SYMBOL_TABLE
"I01"	DB 1	FB 1	// STD - Ilot : DB D'INSTANCE DU FB1
"I02"	DB 2	FB 2	// FACILITY: INSTANCE DB FOR MMC CONTROL (FB2)
"I03"	DB 3	FB 3
"I04"	DB 4	FB 4	// FACILITY: INSTANCE DB FOR COMMUNICATION / DB D'INSTANCE POUR LA COMMUNICATION
"CDIV"	DB 69	DB 69	// FACILITY: DIVERSITIES CODES TABLE / TABLE CODES DIVERSITES
"SFM_DB"	DB 75	FB 20	// Bloque de diagnóstico para Notificar errores de sistema
"SFM_GLOBAL_DB"	DB 76	DB 76	// Bloque de diagnóstico para Notificar errores de sistema
"SFM_PN"	DB 77	DB 77	// PROFINET DIAGNOSTIC FUNCTION EDITING DB FOR IHMP
"SIP1"	DB 89	DB 89	// SIPTOL EXCHANGES DATAS / TABLE D'ECHANGES SIPTOL
"PILE"	DB 90	DB 90	// FACILITY: FIFO STORAGE / PILE DE STOCKAGE
"IDENT"	DB 93	DB 93	// RFID DATAS / IDENTIFIANT DYNAMIQUE
"IBD"	DB 95	DB 95	// FACILITY: DATA BASE DB / DB BASE DE DONNEE
"IIT"	DB 96	DB 96	// FACILITY: PART TABLE / DB TABLE PIECE
"IG"	DB 99	DB 99	// FACILITY: GLOBAL DB / DB GLOBAL
"Z1"	DB 100	FB 100	// ZONE 1: ZONE CONTROL / GESTION ZONE
"Z1A0L"	DB 109	FB 109	// A0 LANCEMENT INSTANCE DATA BLOC / BLOC DE DONNEES INSTANCE A0 LANCEMENT
"Z1A0"	DB 110	FB 110	// A0 MONTAGE INSTANCE DATA BLOC / BLOC DE DONNEES INSTANCE A0 MONTAGE
"Z1A1"	DB 111	FB 111	// A1 OP_BPVAL INSTANCE DATA BLOC / BLOC DE DONNEES INSTANCE A1 OP_BPVAL
"Z1A2"	DB 112	FB 112	// A2 OP_BPVAL INSTANCE DATA BLOC / BLOC DE DONNEES INSTANCE A2 OP_BPVAL
"Z1A0M"	DB 115	FB 115
"Z1B0"	DB 120	FB 120
"Z1B1"	DB 121	FB 121	// B1 OP_BPVAL INSTANCE DATA BLOC / BLOC DE DONNEES INSTANCE B1 OP_BPVAL
"Z1B2"	DB 122	FB 122	// B2 OP_BPVAL INSTANCE DATA BLOC / BLOC DE DONNEES INSTANCE B2 OP_BPVAL
"Z1B3"	DB 123	FB 123	// B3 MONTAGE INSTANCE DATA BLOC / BLOC DE DONNEES INSTANCE B3 MONTAGE
"Z1B4"	DB 124	FB 124	// B4 OP_BIMA INSTANCE DATA BLOC / BLOC DE DONNEES INSTANCE B4 OP_BIMA
"Z1B0M"	DB 125	FB 125
"Z1C0"	DB 130	FB 130	// C0 MONTAGE INSTANCE DATA BLOC / BLOC DE DONNEES INSTANCE C0 MONTAGE
"Z1C1"	DB 131	FB 131	// C1 OP_BPVAL INSTANCE DATA BLOC / BLOC DE DONNEES INSTANCE C1 OP_BPVAL
"Z1D0"	DB 140	FB 140	// D0 MONTAGE INSTANCE DATA BLOC / BLOC DE DONNEES INSTANCE D0 MONTAGE
"Z1D1"	DB 141	FB 141	// D1 OP_BIMA INSTANCE DATA BLOC / BLOC DE DONNEES INSTANCE D1 OP_BIMA
"Z1D2"	DB 142	FB 142	// D2 OP_BIMA INSTANCE DATA BLOC / BLOC DE DONNEES INSTANCE D2 OP_BIMA
"Z1D0R"	DB 143	FB 143	// D0 RECALAGE INSTANCE DATA BLOC / BLOC DE DONNEES INSTANCE D0 RECALAGE
"Z1D0V"	DB 144	FB 144	// DB DE INTANCIA DEL FB 144
"Z1T"	DB 198	DB 198	// ZONE1 : Temps Enveloppe Mouvements
"Z1G"	DB 199	DB 199	// ZONE 1: GLOBAL DB
"Z2"	DB 200	FB 200	// DB DE INSTANCIA FB 200
"Z2LG"	DB 210	FB 210	// DB DE INSTANCIA FB 210
"Z2LG1"	DB 211	FB 211	// DB DE INSTANCIA FB 211
"Z2LD"	DB 220	FB 220	// DB DE INSTANCIA FB 220
"Z2LD1"	DB 221	FB 221	// DB DE INSTANCIA FB 221
"Z2T"	DB 298	DB 298	// ZONE2 : Temps Enveloppe Mouvements
"Z2G"	DB 299	DB 299	// ZONE 2: GLOBAL DB
"DB_DATO_LCB_P0PUP"	DB 601	DB 601	// DB DATOS DEL LECTOR DE CODIGO DE BARRA
"DB_DATO_LCB_B0PUP"	DB 602	DB 602
"DB_DATO_LCB_A0PUPI"	DB 603	DB 603
"ITS0"	DB 1100	FB 1100	// ILOT : DB Instance safety management normal task
"ITSZ1_AU_ES_FZ"	DB 1110	FB 1110	// Z1 : DB D'INSTANCE DU FB 1110
"ITSZ1SOP"	DB 1111	FB 1111	// Z1 : DB D'INSTANCE DU FB 1111
"ITSZ2_AU_ES_FZ"	DB 1120	FB 1120	// Z2 : DB D'INSTANCE DU FB 1120
"ITSZ2SOP"	DB 1121	FB 1121	// Z2 : DB D'INSTANCE DU FB 1121
"TSM"	DB 1279	DB 1279	// ILOT : DB Gestion SAFETY Zone ILOT
"F_GLOBDB"	DB 1300	DB 1300	// F_: F_Global_Data Block
"F00290__D0SB___M11"	DB 1301	FB 1300
"F00284__D0SB___M10"	DB 1302	FB 1300
"F00278__D0SB___M09"	DB 1303	FB 1300
"F00272__D0SB___M08"	DB 1304	FB 1300
"F00013_Z1ZBM06"	DB 1314	FB 1300
"F00019_Z1ZBM07"	DB 1315	FB 1300
"F00304_D0A2"	DB 1316	FB 1300
"F00074_M08"	DB 1318	FB 1300
"F00080_M09"	DB 1319	FB 1300
"F00086_M10"	DB 1320	FB 1300
"F00092_M11"	DB 1321	FB 1300
"F00044_M08"	DB 1322	FB 1300
"F00050_M09"	DB 1323	FB 1300
"F00056_M10"	DB 1324	FB 1300
"F00062_M11"	DB 1325	FB 1300
"F00506_B0A2"	DB 1326	FB 1300
"F00454_B0A2"	DB 1327	FB 1300
"F00404_A0A2"	DB 1328	FB 1300
"F00552__LGSB_M08"	DB 1329	FB 1300
"F00560__LGSB_M09"	DB 1330	FB 1300
"F00566__LGSB_M10"	DB 1331	FB 1300
"F00572__LGSB_M11"	DB 1332	FB 1300
"F00632__LDSB_M08"	DB 1333	FB 1300
"F00640__LDSB_M09"	DB 1334	FB 1300
"F00650__LDSB_M10"	DB 1335	FB 1300
"F00660__LDSB_M11"	DB 1336	FB 1300
"Z1MPDEV"	DB 1600	DB 1600	// PALABRA PIEZA ESPECIFICA MARCHA VACIO
"AFF"	DB 1863	DB 1863	// SIEBERT DISPLAY STRING STORAGE / ALMACENAMIENTO MENSAJE VISULIZADOR SIEBERT
"DB_IHM_Wincc"	DB 1962	FB 1962
"DB_PN"	DB 2036	FB 2036	// INSTANCE IO PROFINET DB
"0_01_ILOT"	FB 1	FB 1
"0_02_MMC"	FB 2	FB 2	// FACILITY: BACKUP MANAGEMENT AND DATA RESTITUTION ON EXTERNAL MMC CARD
"0_03_XOP"	FB 3	FB 3	// STD - ILOT :  FB Gestion des MOP ou LOP
"FB SECU"	FB 4	FB 4
"test_vieAPI"	FB 13	FB 13
"SFM_FB"	FB 20	FB 20	// Bloque de diagnóstico para Notificar errores de sistema
"1_00_ZONE_1"	FB 100	FB 100	// ZONE1 : zone management
"1_A0_LANCEMENT"	FB 109	FB 109	// A0 LANCEMENT FUNCTION BLOC / SECTION PROGRAMME A0 LANCEMENT
"1_A0_STAGE"	FB 110	FB 110	// ZONE1 : stage A0 management
"1_A1_OPERATOR"	FB 111	FB 111	// ZONE1 : operator A1 management
"1_A2_OPERATOR"	FB 112	FB 112	// ZONE1 : operator A2 management
"1_A0_MARIAGE"	FB 115	FB 115	// A0 MARIAGE FUNCTION BLOC / SECTION PROGRAMME A0 MARIAGE
"1_B0_STAGE"	FB 120	FB 120	// ZONE1 : stage B0 management
"1_B1_OPERATOR"	FB 121	FB 121	// ZONE1 : operator B1 management
"1_B2_OPERATOR"	FB 122	FB 122	// ZONE1 : operator B2 management
"1_B3_GRIPPER"	FB 123	FB 123	// Bloque de funcion GRIPPER B0
"1_B4_OP_BIMA"	FB 124	FB 124	// B4 OP_BIMA FUNCTION BLOC / SECTION PROGRAMME B4 OP_BIMA
"1_B0_MARIAGE"	FB 125	FB 125	// B0 MARIAGE FUNCTION BLOC / SECTION PROGRAMME B0 MARIAGE
"1_C0_STAGE"	FB 130	FB 130	// ZONE1 : stage C0 management
"1_C1_OPERATOR"	FB 131	FB 131	// ZONE1 : operator C1 management
"1_D0_STAGE"	FB 140	FB 140	// ZONE1 : stage D0 management
"1_D1_OPERATOR"	FB 141	FB 141	// ZONE1 : operator D1 management
"1_D2_OPERATOR"	FB 142	FB 142	// ZONE1 : operator D2 management
"1_D0_RECALAGE"	FB 143	FB 143	// D0 RECALAGE FUNCTION BLOC / SECTION PROGRAMME D0 RECALAGE
"1_D0_VISU"	FB 144	FB 144	// D0 VISU FUNCTION BLOC / SECTION PROGRAMME D0 VISU
"F_TON"	FB 185	FB 185	// F_: Timer Switch On Delay
"F_TOF"	FB 186	FB 186	// F_: Timer Switch Off Delay
"2_00_ZONE_2"	FB 200	FB 200	// ZONE2 : zone management
"2_LG_MONTAGE"	FB 210	FB 210	// LG MONTAGE FUNCTION BLOC / SECTION PROGRAMME LG MONTAGE
"2_LG1_OP_BIMA"	FB 211	FB 211	// LG1 OP_BIMA FUNCTION BLOC / SECTION PROGRAMME LG1 OP_BIMA
"2_LD_MONTAGE"	FB 220	FB 220	// LD MONTAGE FUNCTION BLOC / SECTION PROGRAMME LD MONTAGE
"2_LD1_OP_BIMA"	FB 221	FB 221	// LD1 OP_BIMA FUNCTION BLOC / SECTION PROGRAMME LD1
"TR0"	FB 1000	FB 1000	// ZONE 1 : FB Gestion SAFETY opérateur ilot
"TRZ1SOP"	FB 1010	FB 1010	// ZONE 1 : FB Gestion SAFETY SOP de la zone 1
"TRZ1SOPR"	FB 1011	FB 1011	// Gestion SAFETY des SCR
"TN0"	FB 1100	FB 1100	// ILOT: FB Gestion SAFETY ilot
"TSZ1_AU_ES_FZ"	FB 1110	FB 1110	// ZONE 1 : FB Gestion SAFETY Arrêt d'Urgence (AU) de la zone 1
"TSZ1_SOP"	FB 1111	FB 1111	// ZONE 1 : FB Gestion SAFETY de la Mise en Service (MS) de la zone 1
"TNZ1FZ"	FB 1112	FB 1112	// ZONE 1 : FB Gestion SAFETY des Fermeture Zone (FZ) de la zone 1
"TNZ1SOP"	FB 1113	FB 1113
"TNZ1VAR"	FB 1114	FB 1114	// ZONE 1 : FB Gestion SAFETY des Relais De Ligne (RLV) de la zone 1
"TSZ2_AU_ES_FZ"	FB 1120	FB 1120	// ZONE 2 : FB Gestion SAFETY Arrêt d'Urgence (AU) de la zone 2
"TSZ2_SOP"	FB 1121	FB 1121	// ZONE 2 : FB Gestion SAFETY de la Mise en Service (MS) de la zone 2
"F_IO_CGP"	FB 1300	FB 1300
"F_CTRL_1"	FB 1301	FB 1301
"F_CTRL_2"	FB 1302	FB 1302
"F_DIAG_N"	FB 1303	FB 1303	// F_: Diagnosticbuffer Message with non CPU-Stop
"FITON"	FB 1304	FB 1304
"FIACK_GL"	FB 1305	FB 1305
"BFI_DEVERM"	FB 1600	FB 1600	// Gestion du déverminage d'une table
"BF_MID_Ordre"	FB 1602	FB 1602
"DP_locator"	FB 1649	FB 1649
"TUSEND"	FB 1681	FB 1681	// Send Data via UDP
"TCON"	FB 1685	FB 1685	// Connect
"PUT"	FB 1689	FB 1689	// Write Data to a Remote CPU
"GET"	FB 1690	FB 1690	// Read Data From a Remote CPU
"F_SENDDP"	FB 1692	FB 1692	// F_: Send Data via PROFIBUS DP / PROFINET IO
"F_ACK_GL"	FB 1695	FB 1695	// ACKNOWLEDGE OF ALL PERIPHERALS F / ACQUITTEMENT GLOBAL PERIPH F
"P_SEND"	FB 1698	FB 1698	// Send Data to CP340
"P_RCV"	FB 1699	FB 1699	// Receive Data from CP340
"BFS_BSEC1"	FB 1710	FB 1710
"BFS_AIR1"	FB 1713	FB 1713
"BFS_CRM1"	FB 1714	FB 1714
"BFS_BIMA"	FB 1719	FB 1719
"BF_DEVERM"	FB 1803	FB 1803	// BF STAGE DRY RUN CONTROL / BF GESTION DEVERMINAGE POSTE
"BF_CARACT_SIEBERT"	FB 1856	FB 1856	// SIEBERT DISPLAY MESSAGE CONFIGURATION / MISE EN FORME MESSAGE AFFICHEUR SIEBERT
"BF_RECALAGE2"	FB 1857	FB 1857
"BF_LANCEMENT"	FB 1858	FB 1858	// GESTION LANCEMENT SIPTOL
"BF_AFF SIEBERT (2*13) PN"	FB 1860	FB 1860
"BF_CONF_MACHINE"	FB 1869	FB 1869	// GESTION BASE DE DONNEE CONFIGURATION MACHINE
"BF_CODE_PROCESS"	FB 1870	FB 1870	// GESTION BASE DE DONNEE CODE PROCESS
"BF_DATABASE3"	FB 1871	FB 1871	// DATABASE MANAGEMENT / GESTION BASE DE DONNEES
"BF_IHMCR1"	FB 1876	FB 1876	// BF gérant l'IHM du relais non piloté par l'API mais controlé
"BF_IHMCRM1"	FB 1877	FB 1877	// BF gérant l'IHM du relais de controçle raccordement de masse CRM
"BF_CABRS"	FB 1897	FB 1897	// Barcode Reader / Lecteur de code a barre
"BF_IHMAIR1"	FB 1931	FB 1931	// BF - ZONE : Diagnostic du bloc BFS_IHMAIR
"BF_ZONE_MODE_IHM1"	FB 1932	FB 1932	// Safety_V2: Zone HMI Operating _modes management/Gestion IHM et mode de la zone
"BF_IHMCRM"	FB 1942	FB 1942	// BF gérant l'IHM du relais de controçle raccordement de masse CRM
"BF_IHMBSEC"	FB 1944	FB 1944	// BF - Zx : Diagnostic SAFETY BFS_BSEC
"BF_MODBUS TCPIP SLAVE"	FB 1961	FB 1961	// Esclave Modbus sur CP Ethernet
"BF_IHM_WINCC"	FB 1962	FB 1962	// BF- Gestion images WinCC Flexible
"BF_PFLEX_PUP"	FB 1999	FB 1999	// Pupitre de recodage
"BF_MMC"	FB 2000	FB 2000	// Sauvegarde et restitution mémoire sur carte mémoire externe (MMC)
"BF_MARIAGE_API"	FB 2003	FB 2003	// Gestion des Mariages Pièces
"BF_ILOT"	FB 2004	FB 2004	// BF- Gestion info lié à l'installation ( Ilot )
"BF_IDENT"	FB 2015	FB 2015
"BF_ROBOT"	FB 2016	FB 2016	// Interface API <=> Robot Version 1.2a
"BF_TCY_SUIV"	FB 2019	FB 2019
"BF_CPT_PIECE"	FB 2021	FB 2021	// BF- Compteur de pièce
"BF_DIAG_PROFINET"	FB 2036	FB 2036	// BF- Diagnostic PROFINET IO
"BF_TF_TP"	FB 2037	FB 2037	// TRANSFERENCIA DE TABLA DE MEMORIAS PIEZAS
"BF_FIFO"	FB 2039	FB 2039
"BF_MOUV2P1"	FB 2042	FB 2042	// BF- Gestion d'un mouvement à 2 positions
"Ilot"	FB 10000	FB 10000	// STD - ILOT : FB Gestion de l'ilot
"Mmc"	FB 10001	FB 10001	// STD - ILOT : FB Gestion de la sauvegarde des données sur carte MMC
"0_00_XOP"	FB 10002	FB 10002	// STD - ILOT :  FB Gestion des MOP ou LOP
"Zone_1"	FB 10100	FB 10100	// STD - Z1 : FB Gestion de la zone
"Z1_ch_elec_flex"	FB 10101	FB 10101	// STD - Z1 : Traitement du changement d'électrodes groupé pour un périmètre flex
"R1_robot_manut"	FB 10511	FB 10511	// R1_robot_manut
"P0_plateau_2pos"	FB 10530	FB 10530	// P0_Mtg: Plateau 2 positions
"V0_elevat"	FB 10600	FB 10600	// V0_elevat
"0_00_CYCLE_ILOT"	FC 1	FC 1	// FACILITY: CALL OF FACILITY FB
"GRP EXE"	FC 2	FC 2
"0_11_SECU_FERMEE"	FC 11	FC 11	// STD - Recopie des informations SAFETY zones 1 à 9 pour la sécurité zone fermée
"SFM_FC"	FC 22	FC 22	// Bloque de diagnóstico para Notificar errores de sistema
"1_00_cycle Z1"	FC 100	FC 100	// Définition cyclique zone 1
"2_00_cycleZ2"	FC 200	FC 200	// Définition cyclique zone 1
"0_00_TSSAFETY"	FC 1100	FC 1100	// STD - ILOT : Groupe d'exécution F associé à l'OB32 (tâche normale)
"0_00_TSCYCLE"	FC 1101	FC 1101	// ILOT : Appel des FB hors opérateurs liées à l'ILOT
"AG_SEND"	FC 1698	FC 1698	// AG SEND
"AG_RECV"	FC 1699	FC 1699	// AG RECEIVE
"Badi"	I 0.0	BOOL	// [MOP1]   BP ANNULATION DEFAUTS ILOT
"Bri"	I 0.1	BOOL	// [MOP1]  BP REARMEMENT ILOT
"bmcy"	I 0.2	BOOL	// [MOP1] ZONE 1: BP MARCHE CYCLE
"smm"	I 0.3	BOOL	// [MOP1] ZONE 1: SEL. MARCHE MANUELLE REGLAGE
"sma"	I 0.4	BOOL	// [MOP1] ZONE 1: SEL. MARCHE AUTOMATIQUE
"bmr"	I 0.5	BOOL	// [MOP1] ZONE 1: BP MOUVEMENT RETOUR
"bma"	I 0.6	BOOL	// [MOP1] ZONE 1: BP MOUVEMENT ALLER
"Dclim"	I 1.0	BOOL	// [MOP1] DEFAUT CLIM. (Option)
"CCFRO1"	I 10.0	BOOL	// Z1B[M02] Safety Common Control 1(F-RO)
"CCFRO2"	I 10.1	BOOL	// Z1B[M02] Safety Common Control 2(F-RO)
"LG_CB380V"	I 10.2	BOOL	// Z1B[M02] LG CB CONTROL DISJUNTOR 380V MOTOR
"LD_CB380V"	I 10.4	BOOL	// Z1B[M02] LD CB CONTROL DISJUNTOR 380V MOTOR
"CCB24Z"	I 10.6	BOOL	// Z1B[M02] Elec.Circuit Breake 24V(1-24Z)
"CCB24R"	I 10.7	BOOL	// Z1B[M02] Elec.Circuit Breake 24V(1-24R)
"CP7b"	I 11.3	BOOL	// Presostato A0
"Z1CRM"	I 11.4	BOOL	// Z1B[M03] CONTROL RELAY CRM
"SOP_bmcy"	I 11.5	BOOL	// [SOP1] ZONE 1: BP MARCHE CYCLE
"SOP_bmr"	I 11.6	BOOL	// [SOP1] ZONE 1: BP MOUVEMENT RETOUR
"SOP_bma"	I 11.7	BOOL	// [SOP1] ZONE 1: BP MOUVEMENT ALLER
"BAUI"	I 13.0	BOOL	// Z1B[M06] EGS Facility(MOP)
"Z1BAU1"	I 13.1	BOOL	// [SOP1] SOP1 ARRET D'URGENCE ILOT
"SSZ11"	I 13.2	BOOL	// Z1B[M06] SAFETY ZONE SELECTOR ON 1
"BAUL12"	I 13.4	BOOL	// Z1B[M06] EGS Facility(LOP) 2
"SSZ12"	I 13.6	BOOL	// Z1B[M06] SAFETY ZONE SELECTOR ON 2
"Z1_AU_FRO"	I 24.0	BOOL	// Z1B[M08] SAFETY RELAY F-RO AU
"Z1_KMS"	I 25.0	BOOL	// Z1B[M09] SAFETY RELAY F-RO ES
"A0_CCSOP"	I 40.0	BOOL	// A0SB[M02] CONTROL POWER NORMAL SOP
"A0_CCSOPTR"	I 40.1	BOOL	// A0SB[M02] CONTROL POWER NORMAL SOPTR
"A0_CCB24Z"	I 40.4	BOOL	// A0SB[M02] Elec.Circuit Breake 24V(24Z)
"A0_CCB24R"	I 40.5	BOOL	// A0SB[M02] Elec.Circuit Breake 24V(24R)
"A1VAL"	I 41.0	BOOL	// A0SB[M03] A1 OPERATION BOX 1 PB ON VALIDATION
"A2VAL"	I 41.1	BOOL	// A0SB[M03] A2 OPERATION BOX 2 PB ON VALIDATION
"A1CPOP1"	I 50.0	BOOL	// A0SB[M09] Laser scanner 1 NORMAL 1-1 A1
"A2CPOP1"	I 50.1	BOOL	// A0SB[M09] Laser scanner 1 NORMAL 2-1 A2
"A1CPOP2"	I 50.4	BOOL	// A0SB[M09] Laser scanner 1 NORMAL 1-2 A1
"A2CPOP2"	I 50.5	BOOL	// A0SB[M09] Laser scanner 1 NORMAL 2-2 A2
"A1BAU1"	I 56.0	BOOL	// A0SB[M10] OPERATION BOX EGS NORMAL 1 A1
"A2BAU1"	I 56.1	BOOL	// A0SB[M10] OPERATION BOX EGS NORMAL 1 A2
"A1BAU2"	I 56.4	BOOL	// A0SB[M10] OPERATION BOX EGS NORMAL 2 A1
"A2BAU2"	I 56.5	BOOL	// A0SB[M10] OPERATION BOX EGS NORMAL 2 A2
"A0_SOP_FRO"	I 67.0	BOOL	// A0SB[M12] OPERATOR SAFETY STAGE A0
"B0_CCSOP"	I 70.0	BOOL	// B0SB[M02] CONTROL POWER NORMAL SOP
"B0_CCSOPTR"	I 70.1	BOOL	// B0SB[M02] CONTROL POWER NORMAL SOPTR
"B0_CCB24Z"	I 70.4	BOOL	// B0SB[M02] Elec.Circuit Breake 24V(24Z)
"B0_CCB24R"	I 70.5	BOOL	// B0SB[M02] Elec.Circuit Breake 24V(24R)
"B1VAL"	I 71.0	BOOL	// B0SB[M03] B1 OPERATION BOX 1 PB ON VALIDATION
"B2VAL"	I 71.1	BOOL	// B0SB[M03] B2 OPERATION BOX 2 PB ON VALIDATION
"A0DCZA"	I 71.4	BOOL	// B0SB[M03] Detector Guinche A0 Zona A
"A0DCZB"	I 71.5	BOOL	// B0SB[M03] Detector Guinche A0 Zona B
"B0DCZC"	I 71.6	BOOL	// B0SB[M03] Detector Guinche B0 Zona C
"B0DCZB"	I 71.7	BOOL	// B0SB[M03] Detector Guinche B0 Zona B
"B1CPOP1"	I 80.0	BOOL	// B0SB[M09] Laser scanner 1 NORMAL 1-1 B1
"B2CPOP1"	I 80.1	BOOL	// B0SB[M09] Laser scanner 1 NORMAL 2-1 B2
"B3_OP4BP11"	I 80.2	BOOL	// B0SB[M09] GRIPPER T-STAND 1 BUTTON 1 (OP3)
"B3_OP4BP21"	I 80.3	BOOL	// B0SB[M09] GRIPPER T-STAND 1 BUTTON 2 (OP3)
"B1CPOP2"	I 80.4	BOOL	// B0SB[M09] Laser scanner 1 NORMAL 1-2 B1
"B2CPOP2"	I 80.5	BOOL	// B0SB[M09] Laser scanner 1 NORMAL 2-2 B2
"B3_OP4BP12"	I 80.6	BOOL	// B0SB[M09] GRIPPER T-STAND 1 BUTTON 1 (OP3)
"B3_OP4BP22"	I 80.7	BOOL	// B0SB[M09] GRIPPER T-STAND 1 BUTTON 2 (OP3)
"B1BAU1"	I 86.0	BOOL	// B0SB[M10] OPERATION BOX EGS NORMAL 1 B1
"B2BAU1"	I 86.1	BOOL	// B0SB[M10] OPERATION BOX EGS NORMAL 1 B2
"B3BAU11"	I 86.2	BOOL	// B0SB[M10] GRIPPER OPERATION BOX EGS NORMAL 3 B1
"B1BAU2"	I 86.4	BOOL	// B0SB[M10] OPERATION BOX EGS NORMAL 2 B1
"B2BAU2"	I 86.5	BOOL	// B0SB[M10] OPERATION BOX EGS NORMAL 2 B2
"B3BAU12"	I 86.6	BOOL	// B0SB[M10] GRIPPER OPERATION BOX EGS NORMAL 3 B2
"B0_SOP_FRO"	I 97.0	BOOL	// B0SB[M12] OPERATOR SAFETY STAGE B0
"B0_SOP_FRO 2"	I 98.0	BOOL	// B0SB[M13] OPERATOR SAFETY GRIPPER B3
"A0LLS103"	I 100.0	BOOL	// ZONE1 [A0I10] A0 LOCATOR LH X SLIDE ADVANCED
"A0LLS115"	I 100.1	BOOL	// ZONE1 [A0I10] A0 LOCATOR LH X AXIS DETECT 1
"A0LLS117"	I 100.2	BOOL	// ZONE1 [A0I10] A0 LOCATOR LH X AXIS DETECT 3
"A0LLS107"	I 100.3	BOOL	// ZONE1 [A0I10] A0 LOCATOR LH Y SLIDE ADVANCED
"A0LLS104"	I 100.4	BOOL	// ZONE1 [A0I10] A0 LOCATOR LH X SLIDE RETURNED
"A0LLS116"	I 100.5	BOOL	// ZONE1 [A0I10] A0 LOCATOR LH X AXIS DETECT 2
"A0LLS108"	I 100.7	BOOL	// ZONE1 [A0I10] A0 LOCATOR LH Y SLIDE RETURNED
"A0LLS119"	I 101.0	BOOL	// ZONE1 [A0I11] A0 LOCATOR LH Y AXIS DETECT 1
"A0LLS121"	I 101.1	BOOL	// ZONE1 [A0I11] A0 LOCATOR LH Y AXIS DETECT 3
"A0LLS111"	I 101.2	BOOL	// ZONE1 [A0I11] A0 LOCATOR LH Z SLIDE ADVANCED
"A0LLS123"	I 101.3	BOOL	// ZONE1 [A0I11] A0 LOCATOR LH Z AXIS DETECT 1
"A0LLS120"	I 101.4	BOOL	// ZONE1 [A0I11] A0 LOCATOR LH Y AXIS DETECT 2
"A0LLS112"	I 101.6	BOOL	// ZONE1 [A0I11] A0 LOCATOR LH Z SLIDE RETURNED
"A0LLS124"	I 101.7	BOOL	// ZONE1 [A0I11] A0 LOCATOR LH Z AXIS DETECT 2
"A0LLS125"	I 102.0	BOOL	// ZONE1 [A0I12] A0 LOCATOR LH Z AXIS DETECT 3
"A0LS001"	I 102.1	BOOL	// ZONE1 [A0I12] A0 CLAMP ADVANCED
"A0LS004"	I 102.2	BOOL	// ZONE1 [A0I12] A0 CLAMP RETURNED 3
"A0LS002"	I 102.5	BOOL	// ZONE1 [A0I12] A0 CLAMP RETURNED 1
"A0LS008"	I 103.0	BOOL	// ZONE1 [A0I13] A0 L38 GAUGE SWING ADVANCED
"A0LS011"	I 103.2	BOOL	// ZONE1 [A0I13] A0 EJECTOR ADVANCED
"A0LS014"	I 103.3	BOOL	// ZONE1 [A0I13] A0 EJECTOR RETURNED 3
"A0LS009"	I 103.4	BOOL	// ZONE1 [A0I13] A0 L38 GAUGE SWING RETURNED 1
"A0LS012"	I 103.6	BOOL	// ZONE1 [A0I13] A0 EJECTOR RETURNED 1
"A0LS016"	I 104.0	BOOL	// ZONE1 [A0I14] A0 GRIPPER SHIFT 1 ADVANCED
"A0LS018"	I 104.1	BOOL	// ZONE1 [A0I14] A0 GRIPPER SHIFT 2 ADVANCED
"A0LS020"	I 104.2	BOOL	// ZONE1 [A0I14] A0 GRIPPER LOCK 1 ADVANCED
"A0LS017"	I 104.4	BOOL	// ZONE1 [A0I14] A0 GRIPPER SHIFT 1 RETURNED
"A0LS019"	I 104.5	BOOL	// ZONE1 [A0I14] A0 GRIPPER SHIFT 2 RETURNED
"A0LS021"	I 104.6	BOOL	// ZONE1 [A0I14] A0 GRIPPER LOCK 1 RETURNED 1
"A0LS022"	I 104.7	BOOL	// ZONE1 [A0I14] A0 GRIPPER LOCK 1 RETURNED 2
"A0LS024"	I 105.0	BOOL	// ZONE1 [A0I15] A0 GRIPPER LOCK 2 ADVANCED
"A0LS027"	I 105.1	BOOL	// ZONE1 [A0I15] A0 MODEL CHANGE 1 ADVANCED
"A0LS030"	I 105.2	BOOL	// ZONE1 [A0I15] A0 MODEL CHANGE 2 ADVANCED
"A0LS025"	I 105.4	BOOL	// ZONE1 [A0I15] A0 GRIPPER LOCK 2 RETURNED 1
"A0LS028"	I 105.5	BOOL	// ZONE1 [A0I15] A0 MODEL CHANGE 1 RETURNED 1
"A0LS031"	I 105.6	BOOL	// ZONE1 [A0I15] A0 MODEL CHANGE 2 RETURNED 1
"A0LS050"	I 106.0	BOOL	// ZONE1 [A0I16] A0 L38 GRIPPER LH DETECT
"A0LS080"	I 106.2	BOOL	// ZONE1 [A0I16] A0 WORK DETECT 1
"A0LS082"	I 106.3	BOOL	// ZONE1 [A0I16] A0 WORK DETECT 3
"A0LS081"	I 106.6	BOOL	// ZONE1 [A0I16] A0 WORK DETECT 2
"A0LS083"	I 106.7	BOOL	// ZONE1 [A0I16] A0 WORK DETECT 4
"A0RLS103"	I 150.0	BOOL	// ZONE1 [A0I20] A0 LOCATOR RH X SLIDE ADVANCED
"A0RLS115"	I 150.1	BOOL	// ZONE1 [A0I20] A0 LOCATOR RH X AXIS DETECT 1
"A0RLS117"	I 150.2	BOOL	// ZONE1 [A0I20] A0 LOCATOR RH X AXIS DETECT 3
"A0RLS107"	I 150.3	BOOL	// ZONE1 [A0I20] A0 LOCATOR RH Y SLIDE ADVANCED
"A0RLS104"	I 150.4	BOOL	// ZONE1 [A0I20] A0 LOCATOR RH X SLIDE RETURNED
"A0RLS116"	I 150.5	BOOL	// ZONE1 [A0I20] A0 LOCATOR RH X AXIS DETECT 2
"A0RLS108"	I 150.7	BOOL	// ZONE1 [A0I20] A0 LOCATOR RH Y SLIDE RETURNED
"A0RLS119"	I 151.0	BOOL	// ZONE1 [A0I21] A0 LOCATOR RH Y AXIS DETECT 1
"A0RLS121"	I 151.1	BOOL	// ZONE1 [A0I21] A0 LOCATOR RH Y AXIS DETECT 3
"A0RLS111"	I 151.2	BOOL	// ZONE1 [A0I21] A0 LOCATOR RH Z SLIDE ADVANCED
"A0RLS123"	I 151.3	BOOL	// ZONE1 [A0I21] A0 LOCATOR RH Z AXIS DETECT 1
"A0RLS120"	I 151.4	BOOL	// ZONE1 [A0I21] A0 LOCATOR RH Y AXIS DETECT 2
"A0RLS112"	I 151.6	BOOL	// ZONE1 [A0I21] A0 LOCATOR RH Z SLIDE RETURNED
"A0RLS124"	I 151.7	BOOL	// ZONE1 [A0I21] A0 LOCATOR RH Z AXIS DETECT 2
"A0RLS125"	I 152.0	BOOL	// ZONE1 [A0I22] A0 LOCATOR RH Z AXIS DETECT 3
"A0LS005"	I 152.2	BOOL	// ZONE1 [A0I22] A0 CLAMP RETURNED 4
"A0LS007"	I 152.3	BOOL	// ZONE1 [A0I22] A0 CLAMP RETURNED 6
"A0LS003"	I 152.5	BOOL	// ZONE1 [A0I22] A0 CLAMP RETURNED 2
"A0LS006"	I 152.6	BOOL	// ZONE1 [A0I22] A0 CLAMP RETURNED 5
"A0LS015"	I 153.3	BOOL	// ZONE1 [A0I23] A0 EJECTOR RETURNED 4
"A0LS010"	I 153.4	BOOL	// ZONE1 [A0I23] A0 L38 GAUGE SWING RETURNED 2
"A0LS013"	I 153.6	BOOL	// ZONE1 [A0I23] A0 EJECTOR RETURNED 2
"A0LS023"	I 154.4	BOOL	// ZONE1 [A0I24] A0 GRIPPER LOCK 1 RETURNED 3
"A0LS026"	I 154.5	BOOL	// ZONE1 [A0I24] A0 GRIPPER LOCK 2 RETURNED 2
"A0LS029"	I 154.6	BOOL	// ZONE1 [A0I24] A0 MODEL CHANGE 1 RETURNED 2
"A0LS032"	I 154.7	BOOL	// ZONE1 [A0I24] A0 MODEL CHANGE 2 RETURNED 2
"A0LS051"	I 155.0	BOOL	// ZONE1 [A0I25] A0 L38 GRIPPER RH DETECT
"A0LS060"	I 156.0	BOOL	// ZONE1 [A0I26] A0 MANUAL CLAMP RETURNED 1
"A0LS084"	I 156.1	BOOL	// ZONE1 [A0I26] A0 PRESENCIA DE PIEZA EN GABARITO TRASERO
"A0LS061"	I 156.4	BOOL	// ZONE1 [A0I26] A0 MANUAL CLAMP RETURNED 2
"A0LS070"	I 156.7	BOOL	// ZONE1 [A0I26] A0 REMORT SYSTEM IN ZONE DETECT
"B0LLS103"	I 200.0	BOOL	// ZONE1 [B0I10] B0 LOCATOR LH X SLIDE ADVANCED
"B0LLS115"	I 200.1	BOOL	// ZONE1 [B0I10] B0 LOCATOR LH X AXIS DETECT 1
"B0LLS117"	I 200.2	BOOL	// ZONE1 [B0I10] B0 LOCATOR LH X AXIS DETECT 3
"B0LLS107"	I 200.3	BOOL	// ZONE1 [B0I10] B0 LOCATOR LH Y SLIDE ADVANCED
"B0LLS104"	I 200.4	BOOL	// ZONE1 [B0I10] B0 LOCATOR LH X SLIDE RETURNED
"B0LLS116"	I 200.5	BOOL	// ZONE1 [B0I10] B0 LOCATOR LH X AXIS DETECT 2
"B0LLS108"	I 200.7	BOOL	// ZONE1 [B0I10] B0 LOCATOR LH Y SLIDE RETURNED
"B0LLS119"	I 201.0	BOOL	// ZONE1 [B0I11] B0 LOCATOR LH Y AXIS DETECT 1
"B0LLS121"	I 201.1	BOOL	// ZONE1 [B0I11] B0 LOCATOR LH Y AXIS DETECT 3
"B0LLS111"	I 201.2	BOOL	// ZONE1 [B0I11] B0 LOCATOR LH Z SLIDE ADVANCED
"B0LLS123"	I 201.3	BOOL	// ZONE1 [B0I11] B0 LOCATOR LH Z AXIS DETECT 1
"B0LLS120"	I 201.4	BOOL	// ZONE1 [B0I11] B0 LOCATOR LH Y AXIS DETECT 2
"B0LLS112"	I 201.6	BOOL	// ZONE1 [B0I11] B0 LOCATOR LH Z SLIDE RETURNED
"B0LLS124"	I 201.7	BOOL	// ZONE1 [B0I11] B0 LOCATOR LH Z AXIS DETECT 2
"B0LLS125"	I 202.0	BOOL	// ZONE1 [B0I12] B0 LOCATOR LH Z AXIS DETECT 3
"B0LS001"	I 202.1	BOOL	// ZONE1 [B0I12] B0 CLAMP ADVANCED
"B0LS004"	I 202.2	BOOL	// ZONE1 [B0I12] B0 CLAMP RETURNED 3
"B0LS002"	I 202.5	BOOL	// ZONE1 [B0I12] B0 CLAMP RETURNED 1
"B0LS006"	I 202.6	BOOL	// ZONE1 [B0I12] B0 CLAMP RETURNED 5
"B0LS008"	I 203.0	BOOL	// ZONE1 [B0I13] B0 L38 GAUGE SWING ADVANCED
"B0LS011"	I 203.1	BOOL	// ZONE1 [B0I13] B0 EJECTOR ADVANCED
"B0LS014"	I 203.2	BOOL	// ZONE1 [B0I13] B0 EJECTOR RETURNED 3
"B0LS016"	I 203.3	BOOL	// ZONE1 [B0I13] B0 OG SHIFT ADVANCED
"B0LS009"	I 203.4	BOOL	// ZONE1 [B0I13] B0 L38 GAUGE SWING RETURNED 1
"B0LS012"	I 203.5	BOOL	// ZONE1 [B0I13] B0 EJECTOR RETURNED 1
"B0LS017"	I 203.7	BOOL	// ZONE1 [B0I13] B0 OG SHIFT RETURNED
"B0LS018"	I 204.0	BOOL	// ZONE1 [B0I14] B0 OG LOCK ADVANCED
"B0LS020"	I 204.1	BOOL	// ZONE1 [B0I14] B0 OG LOCK RETURNED 2
"B0LS050"	I 204.3	BOOL	// ZONE1 [B0I14] B0 L38 GRIPPER DETECT
"B0LS019"	I 204.4	BOOL	// ZONE1 [B0I14] B0 OG LOCK RETURNED 1
"B0LS021"	I 204.5	BOOL	// ZONE1 [B0I14] B0 OG LOCK RETURNED 3
"B0LS022"	I 205.0	BOOL	// ZONE1 [B0I15] B0 GRIPPER LOCK ADVANCED
"B0LS025"	I 205.1	BOOL	// ZONE1 [B0I15] B0 MODEL CHANGE 1 ADVANCED
"B0LS028"	I 205.2	BOOL	// ZONE1 [B0I15] B0 MODEL CHANGE 2 ADVANCED
"B0LS031"	I 205.3	BOOL	// ZONE1 [B0I15] B0 MODEL CHANGE 3 ADVANCED
"B0LS023"	I 205.4	BOOL	// ZONE1 [B0I15] B0 GRIPPER LOCK RETURNED
"B0LS026"	I 205.5	BOOL	// ZONE1 [B0I15] B0 MODEL CHANGE 1 RETURNED
"B0LS029"	I 205.6	BOOL	// ZONE1 [B0I15] B0 MODEL CHANGE 2 RETURNED 1
"B0LS032"	I 205.7	BOOL	// ZONE1 [B0I15] B0 MODEL CHANGE 3 RETURNED 1
"B0LS080"	I 206.0	BOOL	// ZONE1 [B0I16] B0 WORK DETECT 1
"CP7b_B0"	I 206.3	BOOL	// Presostato - B0
"B0LS081"	I 206.4	BOOL	// ZONE1 [B0I16] B0 WORK DETECT 2
"B0RLS103"	I 250.0	BOOL	// ZONE1 [B0I20] B0 LOCATOR RH X SLIDE ADVANCED
"B0RLS115"	I 250.1	BOOL	// ZONE1 [B0I20] B0 LOCATOR RH X AXIS DETECT 1
"B0RLS117"	I 250.2	BOOL	// ZONE1 [B0I20] B0 LOCATOR RH X AXIS DETECT 3
"B0RLS107"	I 250.3	BOOL	// ZONE1 [B0I20] B0 LOCATOR RH Y SLIDE ADVANCED
"B0RLS104"	I 250.4	BOOL	// ZONE1 [B0I20] B0 LOCATOR RH X SLIDE RETURN
"B0RLS116"	I 250.5	BOOL	// ZONE1 [B0I20] B0 LOCATOR RH X AXIS DETECT 2
"B0RLS108"	I 250.7	BOOL	// ZONE1 [B0I20] B0 LOCATOR RH Y SLIDE RETURNED
"B0RLS119"	I 251.0	BOOL	// ZONE1 [B0I21] B0 LOCATOR RH Y AXIS DETECT 1
"B0RLS121"	I 251.1	BOOL	// ZONE1 [B0I21] B0 LOCATOR RH Y AXIS DETECT 3
"B0RLS111"	I 251.2	BOOL	// ZONE1 [B0I21] B0 LOCATOR RH Z SLIDE ADVANCED
"B0RLS123"	I 251.3	BOOL	// ZONE1 [B0I21] B0 LOCATOR RH Z AXIS DETECT 1
"B0RLS120"	I 251.4	BOOL	// ZONE1 [B0I21] B0 LOCATOR RH Y AXIS DETECT 2
"B0RLS112"	I 251.6	BOOL	// ZONE1 [B0I21] B0 LOCATOR RH Z SLIDE RETURNED
"B0RLS124"	I 251.7	BOOL	// ZONE1 [B0I21] B0 LOCATOR RH Z AXIS DETECT 2
"B0RLS125"	I 252.0	BOOL	// ZONE1 [B0I21] B0 LOCATOR RH Z AXIS DETECT 3
"B0LS005"	I 252.2	BOOL	// ZONE1 [B0I22] B0 CLAMP RETURNED 4
"B0LS003"	I 252.5	BOOL	// ZONE1 [B0I22] B0 CLAMP RETURNED 2
"B0LS007"	I 252.6	BOOL	// ZONE1 [B0I22] B0 CLAMP RETURNED 6
"B0LS010"	I 253.4	BOOL	// ZONE1 [B0I23] B0 L38 GAUGE SWING RETURNED 2
"B0LS013"	I 253.5	BOOL	// ZONE1 [B0I23] B0 EJECTOR RETURNED 2
"B0LS015"	I 253.6	BOOL	// ZONE1 [B0I23] B0 EJECTOR RETURNED 4
"B0LS051"	I 253.7	BOOL	// ZONE1 [B0I23] B0 L38 GRIPPER DETECT
"B0LS024"	I 254.4	BOOL	// ZONE1 [B0I24] B0 GRIPPER LOCK RETURNED 2
"B0LS027"	I 254.5	BOOL	// ZONE1 [B0I24] B0 MODEL CHANGE 1 RETURNED 2
"B0LS030"	I 254.6	BOOL	// ZONE1 [B0I24] B0 MODEL CHANGE 2 RETURNED 2
"B0LS033"	I 254.7	BOOL	// ZONE1 [B0I24] B0 MODEL CHANGE 3 RETURNED 2
"B0LS060"	I 255.0	BOOL	// ZONE1 [B0I25] B0 MANUAL CLAMP RETURNED 1
"B0LS062"	I 255.1	BOOL	// ZONE1 [B0I25] B0 MANUAL CLAMP RETURNED 3
"B0LS064"	I 255.2	BOOL	// ZONE1 [B0I25] B0 MANUAL CLAMP RETURNED 5
"B0LS066"	I 255.3	BOOL	// ZONE1 [B0I25] B0 MANUAL CLAMP RETURNED 7
"B0LS061"	I 255.4	BOOL	// ZONE1 [B0I25] B0 MANUAL CLAMP RETURNED 2
"B0LS063"	I 255.5	BOOL	// ZONE1 [B0I25] B0 MANUAL CLAMP RETURNED 4
"B0LS065"	I 255.6	BOOL	// ZONE1 [B0I25] B0 MANUAL CLAMP RETURNED 6
"B0LS067"	I 255.7	BOOL	// ZONE1 [B0I25] B0 MANUAL CLAMP RETURNED 8
"B0LS082"	I 256.0	BOOL	// ZONE1 [B0I26] B0 WORK DETECT 3
"B0LS083"	I 256.4	BOOL	// ZONE1 [B0I26] B0 WORK DETECT 4
"B0LS070"	I 256.7	BOOL	// ZONE1 [B0I26] B0 REMOTE SYSTEM IN ZONE DETECT - Presencia de Griper
"D0_CCFRO1"	I 270.0	BOOL	// D0SB[M02] F-RO1 CONTROL
"D0_CCFRO2"	I 270.1	BOOL	// D0SB[M02] F-RO2 CONTROL
"D0_CCFRO3"	I 270.2	BOOL	// D0SB[M02] F-RO3 CONTROL
"C0DPP1"	I 270.3	BOOL	// D0SB [M02] C0 PART PRESENCE DETECTOR 1
"D0_CCB24Z"	I 270.4	BOOL	// D0SB[M02] CB 24V CONTROL (1-24Z)
"D0_CCB24R"	I 270.5	BOOL	// D0SB[M02] CB 24V CONTROL (2-24R)
"C0DPP2"	I 270.6	BOOL	// D0SB [M02] C0 PART PRESENCE DETECTOR 2
"D0DPG"	I 270.7	BOOL	// D0: DETECTOR PRESENCIA DE GUINCHE
"C1_OP1VAL"	I 271.0	BOOL	// D0SB[M03] C1 OPERATION BOX 1 PB ON VALIDATION
"D0DPP7"	I 271.4	BOOL	// D0SB[M03] D0 PART PRESENCE DETECTOR 7 - CARRO EN POSICION
"C0DCZD"	I 271.5	BOOL	// D0SB[M03] Detector Guinche C0 Zona D
"C0DCZC"	I 271.6	BOOL	// D0SB[M03] Detector Guinche C0 Zona C
"D1BAU1"	I 272.0	BOOL	// D0SB[M08] OPERATION BOX EGS NORMAL 1 D1
"D2BAU1"	I 272.1	BOOL	// D0SB[M08] OPERATION BOX EGS NORMAL 1 D2
"D1BAU2"	I 272.4	BOOL	// D0SB[M08] OPERATION BOX EGS NORMAL 2 D1
"D2BAU2"	I 272.5	BOOL	// D0SB[M08] OPERATION BOX EGS NORMAL 2 D2
"D1_OP1BP11"	I 278.0	BOOL	// D0SB[M09] T-STAND 1 BUTTON 1 (OP1)
"D1_OP1BP21"	I 278.1	BOOL	// D0SB[M09] T-STAND 1 BUTTON 2 (OP1)
"D2_OP2BP11"	I 278.2	BOOL	// D0SB[M09] T-STAND 2 BUTTON 1 (OP2)
"D2_OP2BP21"	I 278.3	BOOL	// D0SB[M09] T-STAND 2 BUTTON 2 (OP2)
"D1_OP1BP12"	I 278.4	BOOL	// D0SB[M09] T-STAND 1 BUTTON 1 (OP1)
"D1_OP1BP22"	I 278.5	BOOL	// D0SB[M09] T-STAND 1 BUTTON 2 (OP1)
"D2_OP2BP12"	I 278.6	BOOL	// D0SB[M09] T-STAND 2 BUTTON 1 (OP2)
"D2_OP2BP22"	I 278.7	BOOL	// D0SB[M09] T-STAND 2 BUTTON 2 (OP2)
"D0_IFRO1"	I 295.0	BOOL	// D0SB[M12] SAFETY  COMMON  1   (FRO-1 - SC3)
"D0_IFRO2"	I 296.0	BOOL	// D0SB[M13] SAFETY  COMMON  2   (FRO-2 - SC4)
"D0_IFRO3"	I 297.0	BOOL	// D0SB[M14] SAFETY  COMMON  3   (FRO-3 - SC5)
"D01DPP1"	I 300.0	BOOL	// ZONE1 [D0E1] D0 PART PRESENCE DETECTOR 1
"D01DPP2"	I 300.1	BOOL	// ZONE1 [D0E1] D0 PART PRESENCE DETECTOR 2
"D01DPP3"	I 300.2	BOOL	// ZONE1 [D0E1] D0 PART PRESENCE DETECTOR 3
"D01DPP4"	I 300.3	BOOL	// ZONE1 [D0E1] D0 PART PRESENCE DETECTOR 4
"D01DPP5"	I 300.4	BOOL	// ZONE1 [D0E1] D0 PART DIVERSITY DETECTOR 1
"D01DPP6"	I 300.5	BOOL	// ZONE1 [D0E1] D0 PART DIVERSITY DETECTOR 2
"D01DPP7"	I 301.0	BOOL	// ZONE1 [D0E1] D0 POCAYOKE CAZOLETA IZQUIERDA
"D01DPP8"	I 301.1	BOOL	// ZONE1 [D0E1] D0 POCAYOKE CAZOLETA DERECHA
"D01DRPL11"	I 302.0	BOOL	// ZONE1 [D0E2] D0 PIN CLAMP RETURNED 1
"D01DAPL11"	I 302.1	BOOL	// ZONE1 [D0E2] D0 PIN CLAMP ADVANCED 1
"D01DRPL12"	I 302.2	BOOL	// ZONE1 [D0E2] D0 PIN CLAMP RETURNED 2
"D01DAPL12"	I 302.3	BOOL	// ZONE1 [D0E2] D0 PIN CLAMP ADVANCED 2
"D01DRSR21"	I 302.4	BOOL	// ZONE1 [D0E2] D0 CLAMP RETURNED 1
"D01DASR21"	I 302.5	BOOL	// ZONE1 [D0E2] D0 CLAMP ADVANCE 1
"D01DRSR22"	I 302.6	BOOL	// ZONE1 [D0E2] D0 CLAMP RETURNED 2
"D01DASR22"	I 302.7	BOOL	// ZONE1 [D0E2] D0 CLAMP ADVANCE 2
"D01DRSR23"	I 303.0	BOOL	// ZONE1 [D0E2] D0 CLAMP RETURNED 3
"D01DASR23"	I 303.1	BOOL	// ZONE1 [D0E2] D0 CLAMP ADVANCE 3
"D01DRSR24"	I 303.2	BOOL	// ZONE1 [D0E2] D0 CLAMP RETURNED 4
"D01DASR24"	I 303.3	BOOL	// ZONE1 [D0E2] D0 CLAMP ADVANCE 4
"CP7b_D0"	I 303.4	BOOL	// Presostato - D0
"A01DPP1"	I 400.0	BOOL	// ZONE1 [A0E1] A0 PART PRESENCE DETECTOR 1
"A01DPP2"	I 400.1	BOOL	// ZONE1 [A0E1] A0 PART PRESENCE DETECTOR 2
"A01DPP3"	I 400.2	BOOL	// ZONE1 [A0E1] A0 PART PRESENCE DETECTOR 3
"A01DASR22"	I 400.3	BOOL	// ZONE1 [A0E1] CLAMP MANUAL SR22 AVANZADO
"A01DPP7"	I 400.4	BOOL	// ZONE1 [A0E1] A0 PART PRESENCE DETECTOR 7
"A01DPP8"	I 400.5	BOOL	// ZONE1 [A0E1] A0 PART PRESENCE DETECTOR 8
"RES1"	I 400.6	BOOL	// ZONE1 [A0E1] A0 MANUAL CLAMP ADVANCED 1
"RES2"	I 400.7	BOOL	// ZONE1 [A0E1] A0 MANUAL CLAMP ADVANCED 2
"A01DRSR11"	I 402.0	BOOL	// ZONE1 [A0E2] A0 CLAMP RETURNED 1
"A01DASR11"	I 402.1	BOOL	// ZONE1 [A0E2] A0 CLAMP ADVANCED 1
"A01DRSR12"	I 402.2	BOOL	// ZONE1 [A0E2] A0 CLAMP RETURNED 2
"A01DASR12"	I 402.3	BOOL	// ZONE1 [A0E2] A0 CLAMP ADVANCED 2
"A01DRSR13"	I 402.4	BOOL	// ZONE1 [A0E2] A0 CLAMP RETURNED 3
"A01DASR13"	I 402.5	BOOL	// ZONE1 [A0E2] A0 CLAMP ADVANCED 3
"A01DRSR14"	I 402.6	BOOL	// ZONE1 [A0E2] A0 CLAMP RETURNED 4
"A01DASR14"	I 402.7	BOOL	// ZONE1 [A0E2] A0 CLAMP ADVANCED 4
"A01DRSR15"	I 403.0	BOOL	// ZONE1 [A0E2] A0 CLAMP RETURNED 5
"A01DASR15"	I 403.1	BOOL	// ZONE1 [A0E2] A0 CLAMP ADVANCED 5
"A01DRSR16"	I 403.2	BOOL	// ZONE1 [A0E2] A0 CLAMP RETURNED 6
"A01DASR16"	I 403.3	BOOL	// ZONE1 [A0E2] A0 CLAMP ADVANCED 6
"B01DPP1"	I 450.0	BOOL	// ZONE1 [B0E1] B0 PART PRESENCE DETECTOR 1
"B01DPP2"	I 450.1	BOOL	// ZONE1 [B0E1] B0 PART PRESENCE DETECTOR 2
"B01DPP3"	I 450.2	BOOL	// ZONE1 [B0E1] B0 PART PRESENCE DETECTOR 3
"B01DPP4"	I 450.3	BOOL	// ZONE1 [B0E1] B0 PART PRESENCE DETECTOR 4
"B01DPP5"	I 450.4	BOOL	// ZONE1 [B0E1] B0 PART PRESENCE DETECTOR 5
"B01DPP6"	I 450.5	BOOL	// ZONE1 [B0E1] B0 PART PRESENCE DETECTOR 6
"B01DRSR11"	I 452.0	BOOL	// ZONE1 [B0E2] B0 CLAMP RETURNED 11
"B01DASR11"	I 452.1	BOOL	// ZONE1 [B0E2] B0 CLAMP ADVANCED 11
"B01DRSR12"	I 452.2	BOOL	// ZONE1 [B0E2] B0 CLAMP RETURNED 12
"B01DASR12"	I 452.3	BOOL	// ZONE1 [B0E2] B0 CLAMP ADVANCED 12
"B01DRSR21"	I 452.4	BOOL	// ZONE1 [B0E2] B0 CLAMP RETURNED 21
"B01DASR21"	I 452.5	BOOL	// ZONE1 [B0E2] B0 CLAMP ADVANCED 21
"B01DRSR22"	I 452.6	BOOL	// ZONE1 [B0E2] B0 CLAMP RETURNED 22
"B01DASR22"	I 452.7	BOOL	// ZONE1 [B0E2] B0 CLAMP ADVANCED 22
"B01DRPL31"	I 453.0	BOOL	// ZONE1 [B0E2] B0 PILOTO RETRAIDO 31
"B01DAPL31"	I 453.1	BOOL	// ZONE1 [B0E2] B0 PILOTO AVANZADO 31
"B01DRPL32"	I 453.2	BOOL	// ZONE1 [B0E2] B0 PILOTO RETRAIDO 32
"B01DAPL32"	I 453.3	BOOL	// ZONE1 [B0E2] B0 PILOTO AVANZADO 32
"B01DRPL41"	I 453.4	BOOL	// ZONE1 [B0E2] B0 PILOTO RETRAIDO 41
"B01DAPL41"	I 453.5	BOOL	// ZONE1 [B0E2] B0 PILOTO AVANZADO 41
"B01DRPL42"	I 453.6	BOOL	// ZONE1 [B0E2] B0 PILOTO RETRAIDO 42
"B01DAPL42"	I 453.7	BOOL	// ZONE1 [B0E2] B0 PILOTO AVANZADO 42
"B01DRPL51"	I 460.0	BOOL	// ZONE1 [B0E3] B0 PINCLAMP RETRAIDO 51
"B01DAPL51"	I 460.1	BOOL	// ZONE1 [B0E3] B0 PINCLAMP AVANZADO 51
"B01DRPL52"	I 460.2	BOOL	// ZONE1 [B0E3] B0 PINCLAMP RETRAIDO 52
"B01DAPL52"	I 460.3	BOOL	// ZONE1 [B0E3] B0 PINCLAMP AVANZADO 52
"B01DRSR61"	I 460.4	BOOL	// ZONE1 [B0E3] B0 CLAMP RETURNED 61
"B01DASR61"	I 460.5	BOOL	// ZONE1 [B0E3] B0 CLAMP ADVANCED 61
"B01DRSR62"	I 460.6	BOOL	// ZONE1 [B0E3] B0 CLAMP RETURNED 62
"B01DASR62"	I 460.7	BOOL	// ZONE1 [B0E3] B0 CLAMP ADVANCED 62
"B02DPP7"	I 500.0	BOOL	// ZONE1 [B0E1] B0 GRIPPER PART PRESENCE DETECTOR 7
"B02DPP8"	I 500.1	BOOL	// ZONE1 [B0E1] B0 GRIPPER PART PRESENCE DETECTOR 8
"B02DPP9"	I 500.2	BOOL	// ZONE1 [B0E1] B0 GRIPPER PART PRESENCE DETECTOR 9
"B02DPP10"	I 500.3	BOOL	// ZONE1 [B0E1] B0 GRIPPER PART PRESENCE DETECTOR 10
"B02DRPL11"	I 502.0	BOOL	// ZONE1 [B0E2] B0 GRIPPER SLIDE RETURNED 11
"B02DAPL11"	I 502.1	BOOL	// ZONE1 [B0E2] B0 GRIPPER SLIDE ADVANCED 11
"B02DRPL12"	I 502.2	BOOL	// ZONE1 [B0E2] B0 GRIPPER SLIDE RETURNED 12
"B02DAPL12"	I 502.3	BOOL	// ZONE1 [B0E2] B0 GRIPPER SLIDE ADVANCED 12
"B02DRPL13"	I 502.4	BOOL	// ZONE1 [B0E2] B0 GRIPPER SLIDE RETURNED 13
"B02DAPL13"	I 502.5	BOOL	// ZONE1 [B0E2] B0 GRIPPER SLIDE ADVANCED 13
"B02DRPL14"	I 502.6	BOOL	// ZONE1 [B0E2] B0 GRIPPER SLIDE RETURNED 14
"B02DAPL14"	I 502.7	BOOL	// ZONE1 [B0E2] B0 GRIPPER SLIDE ADVANCED 14
"B02DRPL21"	I 503.0	BOOL	// ZONE1 [B0E2] B0 GRIPPER SLIDE RETURNED 21
"B02DAPL21"	I 503.1	BOOL	// ZONE1 [B0E2] B0 GRIPPER SLIDE ADVANCED 21
"B02DRPL22"	I 503.2	BOOL	// ZONE1 [B0E2] B0 GRIPPER SLIDE RETURNED 22
"B02DAPL22"	I 503.3	BOOL	// ZONE1 [B0E2] B0 GRIPPER SLIDE ADVANCED 22
"B02DRPL31"	I 503.4	BOOL	// ZONE1 [B0E2] B0 GRIPPER PIN CLAMP RETURNED 31
"B02DAPL31"	I 503.5	BOOL	// ZONE1 [B0E2] B0 GRIPPER PIN CLAMP ADVANCED 31
"B02DRPL32"	I 503.6	BOOL	// ZONE1 [B0E2] B0 GRIPPER PIN CLAMP RETURNED 32
"B02DAPL32"	I 503.7	BOOL	// ZONE1 [B0E2] B0 GRIPPER PIN CLAMP ADVANCED 32
"B02DRPL41"	I 504.0	BOOL	// ZONE1 [B0E2] B0 GRIPPER PIN CLAMP RETURNED 41
"B02DAPL41"	I 504.1	BOOL	// ZONE1 [B0E2] B0 GRIPPER PIN CLAMP ADVANCED 41
"B02DRPL42"	I 504.2	BOOL	// ZONE1 [B0E2] B0 GRIPPER PIN CLAMP RETURNED 42
"B02DAPL42"	I 504.3	BOOL	// ZONE1 [B0E2] B0 GRIPPER PIN CLAMP ADVANCED 42
"B02DRSR51"	I 504.4	BOOL	// ZONE1 [B0E2] B0 GRIPPER CLAMP RETURNED 51
"B02DASR51"	I 504.5	BOOL	// ZONE1 [B0E2] B0 GRIPPER CLAMP ADVANCED 51
"B02DRSR52"	I 504.6	BOOL	// ZONE1 [B0E2] B0 GRIPPER CLAMP RETURNED 52
"B02DASR52"	I 504.7	BOOL	// ZONE1 [B0E2] B0 GRIPPER CLAMP ADVANCED 52
"B02DRSR61"	I 505.0	BOOL	// ZONE1 [B0E2] B0 GRIPPER CLAMP RETURNED 61
"B02DASR61"	I 505.1	BOOL	// ZONE1 [B0E2] B0 GRIPPER CLAMP ADVANCED 61
"B02DRSR62"	I 505.2	BOOL	// ZONE1 [B0E2] B0 GRIPPER CLAMP RETURNED 62
"B02DASR62"	I 505.3	BOOL	// ZONE1 [B0E2] B0 GRIPPER CLAMP ADVANCED 62
"B02SL11"	I 505.4	BOOL	// ZONE1 [B0E2] B0 GRIPPER MODEL SELECT L38
"B02SL12"	I 505.5	BOOL	// ZONE1 [B0E2] B0 GRIPPER MODEL SELECT X52
"B02_CVAL"	I 506.0	BOOL	// [B0A2] CONTRO DE COMUN SEGURIDAD
"B02DRPL71"	I 512.0	BOOL	// ZONE1 [B0E4] B0 GRIPPER PIN CLAMP RETURNED 71
"B02DAPL71"	I 512.1	BOOL	// ZONE1 [B0E4] B0 GRIPPER PIN CLAMP ADVANCED 71
"B02DRPL72"	I 512.2	BOOL	// ZONE1 [B0E4] B0 GRIPPER PIN CLAMP RETURNED 72
"B02DAPL72"	I 512.3	BOOL	// ZONE1 [B0E4] B0 GRIPPER PIN CLAMP ADVANCED 72
"B02DRSR81"	I 512.4	BOOL	// ZONE1 [B0E4] B0 GRIPPER CLAMP RETURNED 81
"B02DASR81"	I 512.5	BOOL	// ZONE1 [B0E4] B0 GRIPPER CLAMP ADVANCED 81
"B02DRSR82"	I 512.6	BOOL	// ZONE1 [B0E4] B0 GRIPPER CLAMP RETURNED 82
"B02DASR82"	I 512.7	BOOL	// ZONE1 [B0E4] B0 GRIPPER CLAMP ADVANCED 82
"LGCCFRO1"	I 550.0	BOOL	// [LGSB.M02]: LG F-RO1 CONTROL
"LGCCFRO2"	I 550.1	BOOL	// [LGSB.M02]: LG F-RO2 CONTROL
"LGCCFRO3"	I 550.2	BOOL	// [LGSB.M02]: LG F-RO3 CONTROL
"LGCB380V"	I 550.3	BOOL	// [LGSB.M02]: LG CB CONTROL DISJUNTOR 380V MOTOR
"LGCCB24Z"	I 550.4	BOOL	// [LGSB.M02]: LG CB 24V CONTROL (1-24Z)
"LGCCB24R"	I 550.5	BOOL	// [LGSB.M02]: LG CB 24V CONTROL (2-24R)
"LGKSOP1"	I 550.6	BOOL	// [LGSB.M02]: LG CONTOLE KSOP1
"LGSB_M2_R1"	I 550.7	BOOL	// [LGSB.M02]: RESERVA
"LGSB_M3_R1"	I 551.0	BOOL	// [LGSB.M03]: RESERVA
"LGSB_M3_R2"	I 551.1	BOOL	// [LGSB.M03]: RESERVA
"LGSB_M3_R3"	I 551.2	BOOL	// [LGSB.M03]: RESERVA
"LGSB_M3_R4"	I 551.3	BOOL	// [LGSB.M03]: RESERVA
"CP7b_LG"	I 551.4	BOOL	// [LGSB.M03]: PRESOSTATO DISPOSITIVO LG
"LGSB_M3_R6"	I 551.5	BOOL	// [LGSB.M03]: RESERVA
"LGSM_X52"	I 551.6	BOOL	// [LGSB.M03]: LD SELECCION MODELO X52
"LGSM_X67"	I 551.7	BOOL	// [LGSB.M03]: LD SELECCION MODELO X67
"LG1BAU1"	I 552.0	BOOL	// [LGSB.M08]: LG1 OPERATOR 1 EGS
"LG2BAU1"	I 552.1	BOOL	// [LGSB.M08]: LG2 OPERATOR 2 EGS
"LGSB_M8_R2"	I 552.2	BOOL	// [LGSB.M08]: RESERVA
"LGSB_M8_R3"	I 552.3	BOOL	// [LGSB.M08]: RESERVA
"LG1BP11"	I 560.0	BOOL	// [LGSB.M09]: LG1 T-STAND 1 BUTTON 1 (OP1) - CH1
"LG1BP21"	I 560.1	BOOL	// [LGSB.M09]: LG1 T-STAND 1 BUTTON 2 (OP1) - CH1
"LG2BP11"	I 560.2	BOOL	// [LGSB.M09]: LG2 T-STAND 2 BUTTON 1 (OP2) - CH1
"LG2BP21"	I 560.3	BOOL	// [LGSB.M09]: LG2 T-STAND 2 BUTTON 2 (OP2) - CH1
"LG1BP12"	I 560.4	BOOL	// [LGSB.M09]: LG1 T-STAND 1 BUTTON 1 (OP1) - CH2
"LG1BP22"	I 560.5	BOOL	// [LGSB.M09]: LG1 T-STAND 1 BUTTON 2 (OP1) - CH2
"LG2BP12"	I 560.6	BOOL	// [LGSB.M09]: LG2 T-STAND 2 BUTTON 1 (OP2) - CH2
"LG2BP22"	I 560.7	BOOL	// [LGSB.M09]: LG2 T-STAND 2 BUTTON 2 (OP2) - CH2
"LGSB_M10_R1"	I 566.0	BOOL	// [LGSB.M10]: RESERVA
"LGSB_M10_R2"	I 566.1	BOOL	// [LGSB.M10]: RESERVA
"LGSB_M10_R3"	I 566.2	BOOL	// [LGSB.M10]: RESERVA
"LGSB_M10_R4"	I 566.3	BOOL	// [LGSB.M10]: RESERVA
"LGIFRO1"	I 577.0	BOOL	// [LGSB.M12]: LG SAFETY COMMON 1 (FRO-1 - SC3)
"LGIFRO2"	I 578.0	BOOL	// [LGSB.M13]: LGSAFETY COMMON 2 (FRO-2 - SC4)
"LGIFRO3"	I 579.0	BOOL	// [LGSB.M14]: LGSAFETY COMMON 3 (FRO-3 - SC5)
"LGDPP2"	I 600.0	BOOL	// [LGIM1.LGE11]: LG: DETECTOR PRESENÇA DE PEÇA 2
"LGDPP1"	I 600.1	BOOL	// [LGIM1.LGE11]: LG: DETECTOR PRESENÇA DE PEÇA 1
"LGDRSR1"	I 600.2	BOOL	// [LGIM1.LGE11]: LG: DETECTOR RETROCESO SR1
"LGDASR1"	I 600.3	BOOL	// [LGIM1.LGE11]: LG: DETECTOR AVANCE SR1
"LGDRSR2"	I 600.4	BOOL	// [LGIM1.LGE11]: LG: DETECTOR RETROCESO SR2
"LGDASR2"	I 600.5	BOOL	// [LGIM1.LGE11]: LG: DETECTOR AVANCE SR2
"LGDRSR3"	I 600.6	BOOL	// [LGIM1.LGE11]: LG: DETECTOR RETROCESO SR3
"LGDASR3"	I 600.7	BOOL	// [LGIM1.LGE11]: LG: DETECTOR AVANCE SR3
"LGDRSR4"	I 601.0	BOOL	// [LGIM1.LGE11]: LG: DETECTOR RETROCESO SR4
"LGDASR4"	I 601.1	BOOL	// [LGIM1.LGE11]: LG: DETECTOR AVANCE SR4
"LGDRVU5"	I 601.2	BOOL	// [LGIM1.LGE11]: LG: DETECTOR RETROCESO VU5
"LGDAVU5"	I 601.3	BOOL	// [LGIM1.LGE11]: LG: DETECTOR AVANCE VU5
"LGDRVU6"	I 601.4	BOOL	// [LGIM1.LGE11]: LG: DETECTOR RETROCESO VU6
"LGDAVU6"	I 601.5	BOOL	// [LGIM1.LGE11]: LG: DETECTOR AVANCE VU6
"LGIM1_LGE12_R7"	I 601.6	BOOL	// [LGIM1.LGE12]: RESERVA
"LGIM1_LGE12_R8"	I 601.7	BOOL	// [LGIM1.LGE12]: RESERVA
"LGIM1_LGE13_R1"	I 602.0	BOOL	// [LGIM1.LGE13]: RESERVA
"LGIM1_LGE13_R2"	I 602.1	BOOL	// [LGIM1.LGE13]: RESERVA
"LGIM1_LGE13_R3"	I 602.2	BOOL	// [LGIM1.LGE13]: RESERVA
"LGIM1_LGE13_R4"	I 602.3	BOOL	// [LGIM1.LGE13]: RESERVA
"LGIM1_LGE13_R5"	I 602.4	BOOL	// [LGIM1.LGE13]: RESERVA
"LGIM1_LGE13_R6"	I 602.5	BOOL	// [LGIM1.LGE13]: RESERVA
"LGIM1_LGE13_R7"	I 602.6	BOOL	// [LGIM1.LGE13]: RESERVA
"LGIM1_LGE13_R8"	I 602.7	BOOL	// [LGIM1.LGE13]: RESERVA
"LGDPA"	I 605.0	BOOL	// [LGIM2.LGE21]: LG: DETECTOR POSIÇÃO AVANÇADO
"LGDPR"	I 605.1	BOOL	// [LGIM2.LGE21]: LG: DETECTOR POSIÇÃO RECUADO
"LGDRPLB1"	I 605.2	BOOL	// [LGIM2.LGE21]: LG: DETECTOR CAMBIO DE MASA ABAJO (MIG)
"LGDAPLB1"	I 605.3	BOOL	// [LGIM2.LGE21]: LG: DETECTOR CAMBIO DE MASA ARRIBA (TUCKER)
"LGIM2_LGE21_R5"	I 605.4	BOOL	// [LGIM2.LGE21]: RESERVA
"LGIM2_LGE21_R6"	I 605.5	BOOL	// [LGIM2.LGE21]: RESERVA
"LGIM2_LGE21_R3"	I 605.6	BOOL	// [LGIM2.LGE21]: RESERVA
"DSG_LGM1"	I 605.7	BOOL	// Detector de segurança de giro mesa LVG500
"LGIM2380V"	I 606.0	BOOL	// [LGIM2.LGSM21]: LG: CONTROLE CHAVE LGIM2
"LGIM2_LGSM21_R1"	I 606.1	BOOL	// [LGIM2.LGSM21]: RESERVA
"LGIM2_LGSM21_R2"	I 606.2	BOOL	// [LGIM2.LGSM21]: RESERVA
"LGIM2_LGSM21_R3"	I 606.3	BOOL	// [LGIM2.LGSM21]: RESERVA
"LGIM2_LGSM21_R4"	I 606.4	BOOL	// [LGIM2.LGSM21]: RESERVA
"LGIM2_LGSM21_R5"	I 606.5	BOOL	// [LGIM2.LGSM21]: RESERVA
"LGIM2_LGSM21_R6"	I 606.6	BOOL	// [LGIM2.LGSM21]: RESERVA
"LGIM2_LGSM21_R7"	I 606.7	BOOL	// [LGIM2.LGSM21]: RESERVA
"LDDPP1"	I 620.0	BOOL	// [LDIM1.LDE11]: LD: DETECTOR PRESENÇA DE PEÇA 1
"LDDPP2"	I 620.1	BOOL	// [LDIM1.LDE11]: LD: DETECTOR RECUO SERRAGE A1
"LDDRSR1"	I 620.2	BOOL	// [LDIM1.LDE11]: LD: DETECTOR RETROCESO SR1
"LDDASR1"	I 620.3	BOOL	// [LDIM1.LDE11]: LD: DETECTOR AVANCE SR1
"LDDRSR2"	I 620.4	BOOL	// [LDIM1.LDE11]: LD: DETECTOR RETROCESO SR2
"LDDASR2"	I 620.5	BOOL	// [LDIM1.LDE11]: LD: DETECTOR AVANCE SR2
"LDDRVU3"	I 620.6	BOOL	// [LDIM1.LDE11]: LD: DETECTOR RETROCESO VU3
"LDDAVU3"	I 620.7	BOOL	// [LDIM1.LDE11]: LD: DETECTOR AVANCE VU3
"LDDRSR4"	I 621.0	BOOL	// [LDIM1.LDE12]: LD: DETECTOR RETROCESO SR4
"LDDASR4"	I 621.1	BOOL	// [LDIM1.LDE12]: LD: DETECTOR AVANCE SR4
"LDDRSR5"	I 621.2	BOOL	// [LDIM1.LDE12]: LD: DETECTOR RETROCESO SR5
"LDDASR5"	I 621.3	BOOL	// [LDIM1.LDE12]: LD: DETECTOR AVANCE SR5
"LDDRVU6"	I 621.4	BOOL	// [LDIM1.LDE12]: LD: DETECTOR RETROCESO VU6
"LDDAVU6"	I 621.5	BOOL	// [LDIM1.LDE12]: LD: DETECTOR AVANCE VU6
"LDDRVU7"	I 621.6	BOOL	// [LDIM1.LDE12]: LD: DETECTOR RETROCESO VU7
"LDDAVU7"	I 621.7	BOOL	// [LDIM1.LDE12]: LD: DETECTOR AVANCE VU7
"LDIM1_LDE13_R1"	I 622.0	BOOL	// [LDIM1.LDE13]: RESERVA
"LDIM1_LDE13_R2"	I 622.1	BOOL	// [LDIM1.LDE13]: RESERVA
"LDIM1_LDE13_R3"	I 622.2	BOOL	// [LDIM1.LDE13]: RESERVA
"LDIM1_LDE13_R4"	I 622.3	BOOL	// [LDIM1.LDE13]: RESERVA
"LDIM1_LDE13_R5"	I 622.4	BOOL	// [LDIM1.LDE13]: RESERVA
"LDIM1_LDE13_R6"	I 622.5	BOOL	// [LDIM1.LDE13]: RESERVA
"LDIM1_LDE13_R7"	I 622.6	BOOL	// [LDIM1.LDE13]: RESERVA
"LDIM1_LDE13_R8"	I 622.7	BOOL	// [LDIM1.LDE13]: RESERVA
"LDDPA"	I 625.0	BOOL	// [LGIM2.LGE21]: LG: DETECTOR POSIÇÃO AVANÇADO
"LDDPR"	I 625.1	BOOL	// [LGIM2.LGE21]: LG: DETECTOR POSIÇÃO RECUADO
"LDIM2_LDE21_R1"	I 625.2	BOOL	// [LDIM2.LDE21]: RESERVA
"LDIM2_LDE21_R2"	I 625.3	BOOL	// [LDIM2.LDE21]: RESERVA
"LDIM2_LDE21_R5"	I 625.4	BOOL	// [LDIM2.LDE21]: RESERVA
"DSG_LDM1"	I 625.5	BOOL	// Detector de segurança de giro mesa LVD500
"LDIM2_LDE21_R3"	I 625.6	BOOL	// [LDIM2.LDE21]: RESERVA
"LDIM2_LDE21_R4"	I 625.7	BOOL	// [LDIM2.LDE21]: RESERVA
"LDIM2380V"	I 626.0	BOOL	// [LDIM2.LDSM21]: LD: CONTROLE CHAVE LDIM2
"LDIM2_LDSM21_R1"	I 626.1	BOOL	// [LDIM2.LDSM21]: RESERVA
"LDIM2_LDSM21_R2"	I 626.2	BOOL	// [LDIM2.LDSM21]: RESERVA
"LDIM2_LDSM21_R3"	I 626.3	BOOL	// [LDIM2.LDSM21]: RESERVA
"LDIM2_LDSM21_R4"	I 626.4	BOOL	// [LDIM2.LDSM21]: RESERVA
"LDIM2_LDSM21_R5"	I 626.5	BOOL	// [LDIM2.LDSM21]: RESERVA
"LDIM2_LDSM21_R6"	I 626.6	BOOL	// [LDIM2.LDSM21]: RESERVA
"LDIM2_LDSM21_R7"	I 626.7	BOOL	// [LDIM2.LDSM21]: RESERVA
"LDCCFRO1"	I 630.0	BOOL	// [LDSB.M02]: LD F-RO1 CONTROL
"LDCCFRO2"	I 630.1	BOOL	// [LDSB.M02]: LD F-RO2 CONTROL
"LDCCFRO3"	I 630.2	BOOL	// [LDSB.M02]: LD F-RO3 CONTROL
"LDCB380V"	I 630.3	BOOL	// [LDSB.M02]: LD CB CONTROL DISJUNTOR 380V MOTOR
"LDCCB24Z"	I 630.4	BOOL	// [LDSB.M02]: LD CB 24V CONTROL (1-24Z)
"LDCCB24R"	I 630.5	BOOL	// [LDSB.M02]: LD CB 24V CONTROL (2-24R)
"LDKSOP1"	I 630.6	BOOL	// [LDSB.M02]: LD CONTOLE KSOP1
"LDSB_M2_R3"	I 630.7	BOOL	// [LDSB.M02]: RESERVA
"LDSB_M3_R5SB_M3_R0"	I 631.0	BOOL	// [LDSB.M03]: RESERVA
"LDSB_M3_R5SB_M3_R1"	I 631.1	BOOL	// [LDSB.M03]: RESERVA
"LDSB_M3_R3"	I 631.2	BOOL	// [LDSB.M03]: RESERVA
"LDSB_M3_R4"	I 631.3	BOOL	// [LDSB.M03]: RESERVA
"CP7b_LD"	I 631.4	BOOL	// [LDSB.M03]: PRESOSTATO DISPOSITIVO LD
"LDSB_M3_R5SB_M3_R6"	I 631.5	BOOL	// [LDSB.M03]: RESERVA
"LDSM_X52"	I 631.6	BOOL	// [LDSB.M03]: LD SELECCION MODELO X52
"LDSM_X67"	I 631.7	BOOL	// [LDSB.M03]: LD SELECCION MODELO X67
"LD1BAU1"	I 632.0	BOOL	// [LDSB_M3_R5SB.M08]: LD1 OPERATOR 1 EGS
"LD2BAU"	I 632.1	BOOL	// [LDSB_M3_R5SB.M08]: LD2 OPERATOR 2 EGS
"LDSB_M3_R5SB_M8_R2"	I 632.2	BOOL	// [LDSB.M08]: RESERVA
"LDSB_M3_R5SB_M8_R3"	I 632.3	BOOL	// [LDSB.M08]: RESERVA
"LD1BP11"	I 640.0	BOOL	// [LDSB.M09]: LD1 T-STAND 1 BUTTON 1 (OP1) - CH1
"LD1BP21"	I 640.1	BOOL	// [LDSB.M09]: LD1 T-STAND 1 BUTTON 2 (OP1) - CH1
"LD2BP11"	I 640.2	BOOL	// [LDSB.M09]: LD2 T-STAND 2 BUTTON 1 (OP2) - CH1
"LD2BP21"	I 640.3	BOOL	// [LDSB.M09]: LD2 T-STAND 2 BUTTON 2 (OP2) - CH1
"LD1BP12"	I 640.4	BOOL	// [LDSB.M09]: LD1 T-STAND 1 BUTTON 1 (OP1) - CH2
"LD1BP22"	I 640.5	BOOL	// [LDSB.M09]: LD1 T-STAND 1 BUTTON 2 (OP1) - CH2
"LD2BP12"	I 640.6	BOOL	// [LDSB.M09]: LD2 T-STAND 2 BUTTON 1 (OP2) - CH2
"LD2BP22"	I 640.7	BOOL	// [LDSB.M09]: LD2 T-STAND 2 BUTTON 2 (OP2) - CH2
"LDSB_M10_R1"	I 650.0	BOOL	// [LDSB.M10]: RESERVA
"LDSB_M10_R2"	I 650.1	BOOL	// [LDSB.M10]: RESERVA
"LDSB_M10_R3"	I 650.2	BOOL	// [LDSB.M10]: RESERVA
"LDSB_M10_R4"	I 650.3	BOOL	// [LDSB.M10]: RESERVA
"LDIFRO1"	I 665.0	BOOL	// [LDSB.M12]: LD SAFETY COMMON 1 (FRO-1 - SC3)
"LDIFRO2"	I 666.0	BOOL	// [LDSB.M13]: LD SAFETY COMMON 2 (FRO-2 - SC4)
"LDIFRO3"	I 667.0	BOOL	// [LDSB.M14]: LD SAFETY COMMON 3 (FRO-3 - SC5)
"BA0"	M 0.0	BOOL	// ILOT: Bit toujours à 0
"BA1"	M 0.1	BOOL	// ILOT: Bit toujours à 1 (Mise Au Point)
"Ba1lien"	M 0.2	BOOL	// ILOT: Bit toujours à 1 (Lien dans les réseaux)
"Shunt"	M 0.3	BOOL	// ILOT: Bit  pour shunter des fonction lors de la Mise Au Point
"Perso"	M 0.4	BOOL	// Equation à personnaliser par le programmeur de l'ilot
"Poub"	M 0.5	BOOL	// Bit Poubelle
"Shunt_crucetas"	M 0.6	BOOL
"Sysfroid"	M 0.7	BOOL	// Détection Démarrage ?froid API (OB100)
"Icl010s"	M 1.0	BOOL	// Info clignotement 0,1 seconde
"Icl020s"	M 1.1	BOOL	// Info clignotement 0,2 seconde
"Icl040s"	M 1.2	BOOL	// Info clignotement 0,4 seconde
"Icl050s"	M 1.3	BOOL	// Info clignotement 0,5 seconde
"Icl080s"	M 1.4	BOOL	// Info clignotement 0,8 seconde
"Icl100s"	M 1.5	BOOL	// Info clignotement 1 seconde
"Icl160s"	M 1.6	BOOL	// Info clignotement 1,6 secondes
"Icl200s"	M 1.7	BOOL	// Info clignotement 2 secondes
"TEST1"	M 5.0	BOOL
"S1B0DPIEC_X52"	M 9.0	BOOL	// Defecto de piezxa - dispositivo B0 - modelos X52
"S1B0DPIEC_iap"	M 9.1	BOOL
"Iadf"	M 9.5	BOOL	// Info Annulation Défaut ILOT (SAFETY)
"Ir"	M 9.6	BOOL	// Info Réarmement ILOT (SAFETY)
"Def_maj"	M 9.7	BOOL	// Défaut Majeur ILOT (SAFETY)
"Z1def_maj"	M 10.0	BOOL	// Z1 : Défaut Majeur Zone (SAFETY)
"Z1Iadf"	M 10.1	BOOL	// Z1 : Info Annulation Défaut Zone (SAFETY)
"Z1Ir"	M 10.2	BOOL	// Z1 : Info Réarmement Zone (SAFETY)
"Z1Manu"	M 10.3	BOOL	// Zone 1 Manual Mode
"Z1mdv"	M 10.4	BOOL	// Zona 1: Modo Deverminage
"Z1IAFJ"	M 10.5	BOOL	// Z1: END OF PRODUCTION STOP INFORMATION (SAFETY)
"IHM_X52"	M 11.0	BOOL
"IHM_L38"	M 11.1	BOOL
"IHM_X67"	M 11.2	BOOL
"Z2def_maj"	M 20.0	BOOL	// Z2 : Défaut Majeur Zone (SAFETY)
"Z2Iadf"	M 20.1	BOOL	// Z2 : Info Annulation Défaut Zone (SAFETY)
"Z2Ir"	M 20.2	BOOL	// Z2 : Info Réarmement Zone (SAFETY)
"Z2Manu"	M 20.3	BOOL	// Zone 2 Manual Mode
"Z2mdv"	M 20.4	BOOL	// Zona 2: Modo Deverminage
"Z2IAFJ"	M 20.5	BOOL	// Z2: END OF PRODUCTION STOP INFORMATION (SAFETY)
"A1OPTIME"	M 30.0	BOOL	// Z1:A1OP End of work for dryrun
"A2OPTIME"	M 30.1	BOOL	// Z1:A2OP End of work for dryrun
"B1OPTIME"	M 30.2	BOOL	// Z1:B1OP End of work for dryrun
"B2OPTIME"	M 30.3	BOOL	// Z1:B2OP End of work for dryrun
"A1MFT1"	M 40.0	BOOL	// Z1:A1 End of work 1
"A1MFT2"	M 40.1	BOOL	// Z1:A1 End of work 2
"A1MFT3"	M 40.2	BOOL	// Z1:A1 End of work 3
"A1MFT4"	M 40.3	BOOL	// Z1:A1 End of work 4
"A1MFT5"	M 40.4	BOOL	// Z1:A1 End of work 5
"A2MFT1"	M 40.5	BOOL	// Z1:A2 End of work 1
"A2MFT2"	M 40.6	BOOL	// Z1:A2 End of work 2
"A2MFT3"	M 40.7	BOOL	// Z1:A2 End of work 3
"A2MFT4"	M 41.0	BOOL	// Z1:A2 End of work 4
"A2MFT5"	M 41.1	BOOL	// Z1:A2 End of work 5
"Aux_B1FT2"	M 41.4	BOOL	// Memoria aux de FT2 para controlar defecto de pieza
"Aux_B2FT2"	M 41.5	BOOL	// Memoria aux de FT2 para controlar defecto de pieza
"aux_A1FT2"	M 41.6	BOOL	// Memoria aux de FT2 para controlar defecto de pieza
"aux_A2FT2"	M 41.7	BOOL	// Memoria aux de FT2 para controlar defecto de pieza
"A0.DEF"	M 42.0	BOOL	// DEFECTO MESA A0
"B0.DEF"	M 42.1	BOOL	// DEFECTO DE MESA B0
"D0.DEF"	M 42.3	BOOL	// DEFECTO MESA D0
"DEF.B3"	M 42.4	BOOL	// DEFECTO B3 GRIPPER
"xALAS"	M 42.6	BOOL
"aux_RAZ"	M 45.0	BOOL	// A0: Marca Aux para puesta a cero de Memorias
"aux_RAZ_B0"	M 45.1	BOOL	// B0: Marca Aux para puesta a cero de Memorias
"aux1_pantalla"	M 46.0	BOOL
"aux2_pantalla"	M 46.1	BOOL
"A0CLM_IR"	M 49.0	BOOL	// A0: Clamp Manuales Informacion Retrocedidos
"A0CLM_IA"	M 49.1	BOOL	// A0: Clamp Manual Informacion Avanzado
"B0CLM_IR"	M 49.2	BOOL	// B0: Clamp Manuales Informacion Retrocedidos
"B0CLM_IA"	M 49.3	BOOL	// B0: Clamp Manuales Informacion Avanzados
"B1MFT1"	M 50.0	BOOL	// Z1:B1 End of work 1
"B1MFT2"	M 50.1	BOOL	// Z1:B1 End of work 2
"B1MFT3"	M 50.2	BOOL	// Z1:B1 End of work 3
"B1MFT4"	M 50.3	BOOL	// Z1:B1 End of work 4
"B1MFT5"	M 50.4	BOOL	// Z1:B1 End of work 5
"B2MFT1"	M 50.5	BOOL	// Z1:B2 End of work 1
"B2MFT2"	M 50.6	BOOL	// Z1:B2 End of work 2
"B2MFT3"	M 50.7	BOOL	// Z1:B2 End of work 3
"B2MFT4"	M 51.0	BOOL	// Z1:B2 End of work 4
"B2MFT5"	M 51.1	BOOL	// Z1:B2 End of work 5
"D1MFT1"	M 60.0	BOOL	// Z1:D1 End of work 1
"D1MFT2"	M 60.1	BOOL	// Z1:D1 End of work 2
"D1MFT3"	M 60.2	BOOL	// Z1:D1 End of work 3
"D1MFT4"	M 60.3	BOOL	// Z1:D1 End of work 4
"D1MFT5"	M 60.4	BOOL	// Z1:D1 End of work 5
"D2MFT1"	M 60.5	BOOL	// Z1:D2 End of work 1
"D2MFT2"	M 60.6	BOOL	// Z1:D2 End of work 2
"aux_B0MFT3"	M 61.4	BOOL	// Fin de trabajo 3 para intercambio con gripper
"F_B02DPP8"	M 70.0	BOOL	// IHM FORZADO B02DPP8
"F_B02DPP9"	M 70.1	BOOL	// IHM FORZADO B02DPP9
"F_B02DPP10"	M 70.2	BOOL	// IHM FORZADO B02DPP10
"F_B02DPP7"	M 70.3	BOOL	// IHM FORZADO B02DPP7
"F_B0LS080"	M 70.4	BOOL	// IHM FORZADO B0LS080
"F_B0LS081"	M 70.5	BOOL	// IHM FORZADO B0LS081
"F_B01DPP6"	M 70.6	BOOL	// IHM FORZADO B02DPP6
"F_B01DPP1"	M 70.7	BOOL	// IHM FORZADO B02DPP1
"F_B01DPP5"	M 71.0	BOOL	// IHM FORZADO B02DPP5
"F_B01DPP3"	M 71.1	BOOL	// IHM FORZADO B02DPP3
"F_DPP"	M 71.2	BOOL	// IHM SUMA DE FORZADOS B0DPP
"xMSERFID"	M 75.0	BOOL	// Memoria de que el RFID fue Escrito
"A1CRS"	M 80.0	BOOL
"A2CRS"	M 80.1	BOOL
"B1CRS"	M 80.2	BOOL
"B2CRS"	M 80.3	BOOL
"Mcpx_ack_req"	M 80.7	BOOL
"S1df_A0SOP"	M 100.0	BOOL
"S1df_B0SOP"	M 100.1	BOOL
"S2df_E0SOP"	M 100.2	BOOL
"S2df_J0SOP"	M 100.3	BOOL
"RFID_OK_AUX"	M 100.5	BOOL
"RFID_ESPERA_AUX"	M 100.6	BOOL
"D0SUMDEF"	M 101.0	BOOL	// D0: sumatoria de defectos
"D1DINHIB1"	M 104.4	BOOL	// D1 DEMANDA DE MODIFICACION DE SEGURIDAD
"D1MINHIB"	M 104.5	BOOL	// D1 MEMORIA INHIBICION DE SEGURIDAD
"D1SOPVINH"	M 104.6	BOOL	// D1 LAMPADA SEGURIDAD INACTIVO
"D1VINHIB"	M 104.7	BOOL	// D1 VALIDACION DE MODIFICACION DE SEGURIDAD
"D1ACONF"	M 105.0	BOOL	// D1 AUTHORIZACION DE MODIFICACION DE SEGURIDAD
"D2DINHIB1"	M 105.1	BOOL	// D2 DEMANDA DE MODIFICACION DE SEGURIDAD
"D2MINHIB"	M 105.2	BOOL	// D2 MEMORIA INHIBICION DE SEGURIDAD
"D2SOPVINH"	M 105.3	BOOL	// D2 LAMPADA SEGURIDAD INACTIVO
"D2VINHIB"	M 105.4	BOOL	// D2 VALIDACION DE MODIFICACION DE SEGURIDAD
"D2ACONF"	M 105.5	BOOL	// D2 AUTHORIZACION DE MODIFICACION DE SEGURIDAD
"A0_AT_A1"	M 201.0	BOOL	// A0: OPERATOR A1 WORK AUTORIZATION / AUTORISATION DE TRAVAIL OPERATEUR A1
"A0_ET_A1"	M 201.1	BOOL	// A0: OPERATOR A1 WORK COMPLETION / ENREGISTREMENT DE TRAVAIL OPERATEUR A1
"A0_AT_A2"	M 202.0	BOOL	// A0: OPERATOR A2 WORK AUTORIZATION / AUTORISATION DE TRAVAIL OPERATEUR A2
"A0_ET_A2"	M 202.1	BOOL	// A0: OPERATOR A2 WORK COMPLETION / ENREGISTREMENT DE TRAVAIL OPERATEUR A2
"A0_AT_A3"	M 203.0	BOOL	// A0: OPERATOR A3 WORK AUTORIZATION / AUTORISATION DE TRAVAIL OPERATEUR A3
"A0_ET_A3"	M 203.1	BOOL	// A0: OPERATOR A3 WORK COMPLETION / ENREGISTREMENT DE TRAVAIL OPERATEUR A3
"B0_AT_B1"	M 205.0	BOOL	// B0: OPERATOR B1 WORK AUTORIZATION / AUTORISATION DE TRAVAIL OPERATEUR B1
"B0_ET_B1"	M 205.1	BOOL	// B0: OPERATOR B1 WORK COMPLETION / ENREGISTREMENT DE TRAVAIL OPERATEUR B1
"B0_AT_B2"	M 206.0	BOOL	// B0: OPERATOR B2 WORK AUTORIZATION / AUTORISATION DE TRAVAIL OPERATEUR B2
"B0_ET_B2"	M 206.1	BOOL	// B0: OPERATOR B2 WORK COMPLETION / ENREGISTREMENT DE TRAVAIL OPERATEUR B2
"B3_AT_B4"	M 206.2	BOOL	// B3: OPERATOR B4 WORK COMPLETION / ENREGISTREMENT DE TRAVAIL OPERATEUR B4
"B3_ET_B4"	M 206.3	BOOL	// B3: OPERATOR B4 WORK COMPLETION / ENREGISTREMENT DE TRAVAIL OPERATEUR B4
"C0_AT_C1"	M 207.0	BOOL	// C0: OPERATOR C1 WORK AUTORIZATION / AUTORISATION DE TRAVAIL OPERATEUR C1
"C0_ET_C1"	M 207.1	BOOL	// C0: OPERATOR C1 WORK COMPLETION / ENREGISTREMENT DE TRAVAIL OPERATEUR C1
"C0_AT_C2"	M 208.0	BOOL	// C0: OPERATOR C2 WORK AUTORIZATION / AUTORISATION DE TRAVAIL OPERATEUR C2
"C0_ET_C2"	M 208.1	BOOL	// C0: OPERATOR C2 WORK COMPLETION / ENREGISTREMENT DE TRAVAIL OPERATEUR C2
"C0_AT_C3"	M 210.0	BOOL	// C0: OPERATOR C1 WORK AUTORIZATION / AUTORISATION DE TRAVAIL OPERATEUR C1
"C0_ET_C3"	M 210.1	BOOL	// C0: OPERATOR C1 WORK COMPLETION / ENREGISTREMENT DE TRAVAIL OPERATEUR C1
"B0_AT_B3"	M 211.0	BOOL	// B0: OPERATOR B3 WORK AUTORIZATION / AUTORISATION DE TRAVAIL OPERATEUR B3
"B0_ET_B3"	M 211.1	BOOL	// B0: OPERATOR B3 WORK COMPLETION / ENREGISTREMENT DE TRAVAIL OPERATEUR B3
"B0_AT_B4"	M 212.0	BOOL	// B0: OPERATOR B4 WORK AUTORIZATION / AUTORISATION DE TRAVAIL OPERATEUR B4
"B0_ET_B4"	M 212.1	BOOL	// B0: OPERATOR B4 WORK COMPLETION / ENREGISTREMENT DE TRAVAIL OPERATEUR B4
"B3_SEL_L38"	M 212.2	BOOL	// B3: Seleccion de modelo L38
"B3_SEL_X52"	M 212.3	BOOL	// B3: Seleccion de modelo X52
"D0_AT_D1"	M 213.0	BOOL	// D0: OPERATOR D1 WORK AUTORIZATION / AUTORISATION DE TRAVAIL OPERATEUR D1
"D0_ET_D1"	M 213.1	BOOL	// D0: OPERATOR D1 WORK COMPLETION / ENREGISTREMENT DE TRAVAIL OPERATEUR D1
"D0_AT_D2"	M 214.0	BOOL	// D0: OPERATOR D2 WORK AUTORIZATION / AUTORISATION DE TRAVAIL OPERATEUR D2
"D0_ET_D2"	M 214.1	BOOL	// D0: OPERATOR D2 WORK COMPLETION / ENREGISTREMENT DE TRAVAIL OPERATEUR D2
"B0_SAFETY_RET_L38"	M 215.0	BOOL
"B0_SAFETY_RET_X52"	M 215.1	BOOL
"B0_SAFETY_RET_X67"	M 215.2	BOOL
"LG_AT_LG1"	M 220.0	BOOL	// LG: OPERATOR LG1 WORK AUTORIZATION / AUTORISATION DE TRAVAIL OPERATEUR LG1
"LG_ET_LG1"	M 220.1	BOOL	// LG: OPERATOR LG1 WORK COMPLETION / ENREGISTREMENT DE TRAVAIL OPERATEUR LG1
"LG_AT_LG2"	M 220.2	BOOL	// LG: OPERATOR LG2 WORK AUTORIZATION / AUTORISATION DE TRAVAIL OPERATEUR LG2
"LG_ET_LG2"	M 220.3	BOOL	// LG: OPERATOR LG2 WORK COMPLETION / ENREGISTREMENT DE TRAVAIL OPERATEUR LG2
"LD_AT_LD1"	M 221.0	BOOL	// LD: OPERATOR LD1 WORK AUTORIZATION / AUTORISATION DE TRAVAIL OPERATEUR LD1
"LD_ET_LD1"	M 221.1	BOOL	// LD: OPERATOR LD1 WORK COMPLETION / ENREGISTREMENT DE TRAVAIL OPERATEUR LD1
"LD_AT_LD2"	M 221.2	BOOL	// LD: OPERATOR LD2 WORK AUTORIZATION / AUTORISATION DE TRAVAIL OPERATEUR LD2
"LD_ET_LD2"	M 221.3	BOOL	// LD: OPERATOR LD2 WORK COMPLETION / ENREGISTREMENT DE TRAVAIL OPERATEUR LD2
"MSOKPIS1"	M 222.0	BOOL	// PISTOLA 1 M5 SOLDA OK
"MSOKPIS2"	M 222.1	BOOL	// PISTOLA 2 M5 SOLDA OK
"MSOKPIS3"	M 222.2	BOOL	// PISTOLA 3 M8 SOLDA OK
"MSOKPIS4"	M 222.3	BOOL
"A0_LOCCHANGE"	M 250.0	BOOL	// AUTORIZACION CAMBIO DE POSICION LOCATORS
"A1_LOCCHANGE"	M 250.1	BOOL	// AUTORIZACION OPERADOR 1 CAMBIO DE POSICION LOCATORS
"A2_LOCCHANGE"	M 250.2	BOOL	// AUTORIZACION OPERADOR 2 CAMBIO DE POSICION LOCATORS
"B0_LOCCHANGE"	M 260.0	BOOL	// AUTORIZACION CAMBIO DE POSICION LOCATORS
"B1_LOCCHANGE"	M 260.1	BOOL	// AUTORIZACION OPERADOR 1 CAMBIO DE POSICION LOCATORS
"B2_LOCCHANGE"	M 260.2	BOOL	// AUTORIZACION OPERADOR 2 CAMBIO DE POSICION LOCATORS
"A0_SMD"	M 270.0	BOOL	// A0 - SELECCION MODO DEVERMINAGE DESDE HMI
"B0_SMD"	M 270.1	BOOL	// B0 - SELECCION MODO DEVERMINAGE DESDE HMI
"D0_SMD"	M 270.2	BOOL	// D0 - SELECCION MODO DEVERMINAGE DESDE HMI
"Z1_SDV"	M 270.3	BOOL	// Z1 - SELECCION MODO DEVERMINAGE DESDE HMI
"MDVSEL_X52"	M 270.4	BOOL	// Z1 - SELECCION MODELO X52 PARA MODO DEVERMINAGE
"MDVSEL_L38"	M 270.5	BOOL	// Z1 - SELECCION MODELO L38 PARA MODO DEVERMINAGE
"LG_SMD"	M 270.6	BOOL	// LG - SELECCION MODO DEVERMINAGE DESDE HMI
"LD_SMD"	M 270.7	BOOL	// LD - SELECCION MODO DEVERMINAGE DESDE HMI
"MDVSEL_X67"	M 271.0	BOOL	// Z1 - SELECCION MODELO X67 PARA MODO DEVERMINAGE
"Scaner_cortado"	M 300.0	BOOL	// Scaner cortado en un desplazamiento de locaetor
"MSOLDOKM6"	M 301.1	BOOL	// MEMORIA DE SOLDA OK PISTOLA M6
"MDEC"	M 310.0	BOOL	// Memoria defeito extra curso LVG500
"MDEC_IM2"	M 310.1	BOOL	// Memoria defeito extra curso LVD500
"D0_D1_AT"	M 317.4	BOOL	// Z1: Tool D0 operator work enable D1
"D0_D2_AT"	M 317.5	BOOL	// Z1: Tool D0 operator work enable D2
"D0_D3_AT"	M 317.6	BOOL	// Z1: Tool D0 operator work enable D3
"D0_D4_AT"	M 317.7	BOOL	// Z1: Tool D0 operator work enable D4
"D0_D1_ET"	M 318.0	BOOL	// Z1: Tool D0 operator work completion D1
"D0_D2_ET"	M 318.1	BOOL	// Z1: Tool D0 operator work completion D2
"D0_D3_ET"	M 318.2	BOOL	// Z1: Tool D0 operator work completion D3
"D0_D4_ET"	M 318.3	BOOL	// Z1: Tool D0 operator work completion D4
"A1CRSA0"	M 318.4	BOOL	// A1: SAFETY RESET CONDITION / CONDITION DE REARMEMENT SECURITE
"A2CRSA0"	M 318.5	BOOL	// A2: SAFETY RESET CONDITION / CONDITION DE REARMEMENT SECURITE
"B1CRSB0"	M 318.6	BOOL	// B1: SAFETY RESET CONDITION / CONDITION DE REARMEMENT SECURITE
"B2CRSB0"	M 318.7	BOOL	// B2: SAFETY RESET CONDITION / CONDITION DE REARMEMENT SECURITE
"SCADA"	M 333.0	BOOL
"A0_B0_TROK"	M 400.0	BOOL
"AUX_CAZ_IZQ"	M 401.0	BOOL	// ZONE1 [D0E1] D0 AUXILIAR CAZOLETA IZQUIERDA
"AUX_CAZ_DER"	M 401.1	BOOL	// ZONE1 [D0E1] D0 AUXILIAR CAZOLETA DERECHA
"AUX_CAZ_OK"	M 401.2	BOOL	// ZONE1 [D0E1] D0 AUXILIAR CAZOLETA OK
"S1D0CAZO"	M 401.3	BOOL	// DEFECTO CARGA CAZOLETA
"MANU_D1"	M 450.0	BOOL	// seleccion pupitre manual desde pantalla D1
"MANU_D2"	M 450.1	BOOL	// seleccion pupitre manual desde pantalla D2
"TEMP_ZONO"	M 500.0	BOOL	// TEMP STARTUP TO REMOVE
"M_Val_A0"	M 500.1	BOOL	// Memoria de activacion de validacion unica dispositivo A0
"M_Val_B0"	M 500.2	BOOL	// Memoria de activacion de validacion unica dispositivo B0
"BP_BIM_LD"	M 500.3	BOOL	// AUXILIAR BY PASS BIMANUAL LD
"BP_BIM_LG"	M 500.4	BOOL	// AUXILIAR BY PASS BIMANUAL LG
"aux_A0_Mdroc"	M 501.1	BOOL	// Memoria de Retorrno Origen en Proceso
"aux_B0_Mdroc"	M 501.2	BOOL	// Memoria de Retorrno Origen en Proceso
"aux_C0_Mdroc"	M 501.3	BOOL	// Memoria de Retorrno Origen en Proceso
"aux_D0_Mdroc"	M 501.4	BOOL	// Memoria de Retorrno Origen en Proceso
"BROC_A0"	M 505.0	BOOL	// Retorrno Origen A0
"BROC_B0"	M 505.1	BOOL	// Retorrno Origen B0
"BROC_D0"	M 505.2	BOOL	// Retorrno Origen D0
"BROC_LG"	M 505.3	BOOL	// Retorrno Origen LG
"BROC_LD"	M 505.4	BOOL	// Retorrno Origen LD
"A0_RCLT_L38"	M 505.5	BOOL	// A0 AVISO RETRAER CLAMP GABARITO TRASERO L38
"A0_RCLT_X52"	M 505.6	BOOL	// A0 AVISO RETRAER CLAMP GABARITO TRASERO X52
"A0_RCLD_X52"	M 505.7	BOOL	// A0 AVISO RETRAER CLAMP GABARITO DELANTERO X52
"AUX_DEF_LG"	M 506.0	BOOL	// AUXILIAR DEFECTO LG
"AUX_DEF_LD"	M 506.1	BOOL	// AUXILIAR DEFECTO LD
"XLGCARSOP1"	M 902.0	BOOL	// LG AUXILIAR COMANDO AVANÇO RECUO SOP1
"XLDCARSOP1"	M 903.0	BOOL	// LD AUXILIAR COMANDO AVANÇO RECUO SOP1
"MCROK"	M 959.3	BOOL	// MEMORIA AUX RESULTADO OK DE TODAS AS PISTOLA
"MBPT"	M 959.4	BOOL	// Memória Bypass contador de Tucker
"MDCONT"	M 959.5	BOOL	// Memória defeito contador de Tucker
"MSOLDOKMAS"	M 959.7	BOOL	// MEMORIA SOLDA OK PISTOLA PINO MASSA
"MACT"	M 960.4	BOOL	// Memória auxiliar contador de Tucker FAG0063
"MAHCT"	M 960.5	BOOL	// Memória auxiliar habilita contador de Tucker
"MDFT"	M 960.6	BOOL	// Memória defeito falta de Tucker
"MHAB_M6"	M 960.7	BOOL	// MEMORIA HABILITA CONTADOR M6
"M_CT_OK"	M 999.0	BOOL	// Memoria contador ok
"D1_DEF"	M 1000.0	BOOL	// D1 : Défaut présent dans gestion du sous ensemble
"D2_DEF"	M 1000.1	BOOL	// D2 : Défaut présent dans gestion du sous ensemble
"A0_TYPE CHANGE"	M 1000.6	BOOL	// =1 si hay cambio de modelo
"D0_HMI_SEL_L38"	M 1001.1	BOOL	// D0 Seleccion de modelo L38 desde HMI
"D0_HMI_SEL_L52"	M 1001.2	BOOL	// D0 Seleccion de modelo L52 desde HMI
"D0_HMI_SEL_B52"	M 1001.3	BOOL	// D0 Seleccion de modelo B52 desde HMI
"B0_TYPE CHANGE"	M 1001.4	BOOL	// =1 si hay cambio de modelo
"S1DFCMOD"	M 1001.7	BOOL	// B0: DEFECTO CAMBIO DE MODELO
"M_CT_LVD_ok"	M 1020.0	BOOL	// Memoria de contador ok.
"LGSM_X52_IHMP"	M 1100.0	BOOL	// [LGSB.M03]: LD SELECCION MODELO X52 IHMP
"LGSM_X67_IHMP"	M 1100.1	BOOL	// [LGSB.M03]: LD SELECCION MODELO X67 IHMP
"S1ActR8"	M 2002.0	BOOL	// Z1 : Mot d'action Réserve Rang 8 du Bool / 8th Bool Reserved for Order Word
"S1ActR9"	M 2002.1	BOOL	// Z1 : Mot d'action Réserve Rang 9 du Bool / 9th Bool Reserved for Order Word
"S1ActR10"	M 2002.2	BOOL	// Z1 : Mot d'action Réserve Rang 10 du Bool / 10th Bool Reserved for Order Word
"S1ActR11"	M 2002.3	BOOL	// Z1 : Mot d'action Réserve Rang 11 du Bool / 11th Bool Reserved for Order Word
"S1ActR12"	M 2002.4	BOOL	// Z1 : Mot d'action Réserve Rang 12 du Bool / 12th Bool Reserved for Order Word
"S1ActR13"	M 2002.5	BOOL	// Z1 : Mot d'action Réserve Rang 13 du Bool / 13th Bool Reserved for Order Word
"S1ActR14"	M 2002.6	BOOL	// Z1 : Mot d'action Réserve Rang 14 du Bool / 14th Bool Reserved for Order Word
"S1ActR15"	M 2002.7	BOOL	// Z1 : Mot d'action Réserve Rang 15 du Bool / 15th Bool Reserved for Order Word
"S1BLZ"	M 2003.0	BOOL	// Z1:  Demande de Blocage Zone / Demand of Blocking Zone
"S1DD0"	M 2003.1	BOOL	// Z1 : Demamde de documentation / Demand of documentation
"S1DPR"	M 2003.2	BOOL	// Z1 : Demande de préventif / Demande of preventive
"S1RAZ"	M 2003.3	BOOL	// Z1 : Demande de RAz compteur / Demand of meter reset
"S1ITR"	M 2003.4	BOOL	// Z1 : InfoTemps Requis Zone / Request time zone
"S1ActR5"	M 2003.5	BOOL	// Z1 : Mot d'action Réserve Rang 5 du Bool / 5th Bool Reserved for Order Word
"S1ActR6"	M 2003.6	BOOL	// Z1 : Mot d'action Réserve Rang 6 du Bool / 6th Bool Reserved for Order Word
"S1ActR7"	M 2003.7	BOOL	// Z1 : Mot d'action Réserve Rang 7 du Bool / 7th Bool Reserved for Order Word
"S1ETAR8"	M 2004.0	BOOL	// Z1 : Mot d'Etat Réserve Rang 8 du Bool / 8th Bool Reserved for Status Word
"S1ETAR9"	M 2004.1	BOOL	// Z1 : Mot d'Etat Réserve Rang 9 du Bool / 9th Bool Reserved for Status Word
"S1ETAR10"	M 2004.2	BOOL	// Z1 : Mot d'Etat Réserve Rang 10 du Bool / 10th Bool Reserved for Status Word
"S1ETAR11"	M 2004.3	BOOL	// Z1 : Mot d'Etat Réserve Rang 11 du Bool / 11th Bool Reserved for Status Word
"S1ETAR12"	M 2004.4	BOOL	// Z1 : Mot d'Etat Réserve Rang 12 du Bool / 12th Bool Reserved for Status Word
"S1ETAR13"	M 2004.5	BOOL	// Z1 : Mot d'Etat Réserve Rang 13 du Bool / 13th Bool Reserved for Status Word
"S1ETAR14"	M 2004.6	BOOL	// Z1 : Mot d'Etat Réserve Rang 14 du Bool / 14th Bool Reserved for Status Word
"S1ETAR15"	M 2004.7	BOOL	// Z1 : Mot d'Etat Réserve Rang 15 du Bool / 15th Bool Reserved for Status Word
"S1APP"	M 2005.0	BOOL	// Z1 : Arret Pour Panne / Stop for Fault
"S1APE"	M 2005.1	BOOL	// Z1 : Arret Pour Exploitation / Stop for Exploitation
"S1APF"	M 2005.2	BOOL	// Z1 : Arret Pour Fabrication / Stop For Manufacturing
"S1ETAR3"	M 2005.3	BOOL	// Z1 : Mot d'Etat Réserve Rang 3 du Bool / 3rd Bool Reserved for Status Word
"S1ETAR4"	M 2005.4	BOOL	// Z1 : Mot d'Etat Réserve Rang 4 du Bool / 4th Bool Reserved for Status Word
"S1ETAR5"	M 2005.5	BOOL	// Z1 : Mot d'Etat Réserve Rang 5 du Bool / 5th Bool Reserved for Status Word
"S1ETAR6"	M 2005.6	BOOL	// Z1 : Mot d'Etat Réserve Rang 6 du Bool / 6th Bool Reserved for Status Word
"S1ETAR7"	M 2005.7	BOOL	// Z1 : Mot d'Etat Réserve Rang 7 du Bool / 7th Bool Reserved for Status Word
"MSP1P2P3"	MW 952	WORD	// MEMORIA DE RESULTADO DE SOMA PISTOLAS 1,2 E 3
"MCONT_M6"	MW 954	WORD	// MEMORIA CONTADOR M5
"MCONT_MASS"	MW 956	WORD	// Memoria contagem pino massa
"MACT1"	MW 961	WORD	// CONTADOR DE TUCKER PISTOLA 1 M5 FAG0031
"MACT2"	MW 963	WORD	// CONTADOR DE TUCKER PISTOLA 2 M5 FAG0031
"MACT3"	MW 965	WORD	// CONTADOR DE TUCKER PISTOLA 3 M8 FAG0031
"MACT4"	MW 967	WORD	// CONTADOR DE TUCKER PISTOLA 4 M6 FAG0031
"MAUXBF"	MW 969	WORD	// MEMORIA AUXILIAR BUFFER CONTADOR PISTOLA 1 E 2
"MAUXBF1"	MW 971	WORD	// MEMORIA AUXILIAR BUFFER PISTOLA 3 E 4
"MSTPIST"	MW 973	WORD	// SOMA DE TODAS AS PISTOLA
"MCONT1"	MW 975	WORD	// MEMORIA DE CONTADOR DE TUCKER PISTOLA 1
"MCONT"	MW 977	WORD	// MEMORIA DE CONTADOR DE TUCKER PISTOLA 1 M6
"MCONT3"	MW 979	WORD	// MEMORIA DE CONTADOR DE TUCKER PISTOLA 4
"MSP1E2"	MW 981	WORD	// MEMORIA SOMA PISTOLA 1 E 2
"MSTP"	MW 983	WORD	// MEMORIA SOMA TODAS AS PISTOLA
"MSP2E3"	MW 985	WORD	// Memória soma da pistola 2 e 3 LVG500
"S_Vieapi"	MW 2000	WORD	// Mot de vie Api / Life Word PLC
"S1ACT"	MW 2002	WORD	// Z1 : Mot D'action SMP / SMP order Word
"S1ETA"	MW 2004	WORD	// Z1 : Mot détat SMP / SMP Status Word
"S1PRO1"	MW 2006	INT	// Z1 : Compteur de production / Meter of production
"S1TCY"	MW 2008	WORD	// Z1 : Numéro de cycle / Cycle Number
"S1TCP"	MW 2010	WORD	// Z1 : Temps de cycle Propre / Proper Cycle Time
"S1TCT"	MW 2012	WORD	// Z1 : Temps de cycle Total  / Cycle Time
"CYCL_EXC"	OB 1	OB 1	// Cycle Execution
"CYC_INT4"	OB 34	OB 34	// Cyclic Interrupt 4
"I/O_FLT1"	OB 82	OB 82	// I/O Point Fault 1
"I/O_FLT2"	OB 83	OB 83	// I/O Point Fault 2
"OBNL_FLT"	OB 85	OB 85	// OB Not Loaded Fault
"RACK_FLT"	OB 86	OB 86	// Loss of Rack Fault
"COMPLETE RESTART"	OB 100	OB 100	// Complete Restart
"PROG_ERR"	OB 121	OB 121	// Programming Error
"MOD_ERR"	OB 122	OB 122	// Module Access Error
"Vadi"	Q 0.0	BOOL	// [MOP1] VOYANT ANNULATION DEFAUT INSTALLATION
"vmcy1"	Q 0.1	BOOL	// [MOP1] ZONE 1:VOYANT MARCHE CYCLE
"Raop"	Q 0.3	BOOL	// [MOP1] RELAIS APPEL OPERATEUR
"AlaS"	Q 1.0	BOOL	// ZONE 1 : Alarma Sonora
"AlaL"	Q 1.1	BOOL	// ZONE 1 : Alarma Luminosa
"SOP_vmcy"	Q 12.0	BOOL	// [SOP1] ZONE 1:VOYANT MARCHE CYCLE
"Z1AU"	Q 19.0	BOOL	// Z1B[M07] SAFETY LEVEL OUTPUT AU
"Z1ES"	Q 19.1	BOOL	// Z1B[M07] SAFETY LEVEL OUTPUT ES
"EV7b"	Q 19.3	BOOL	// Z1B[M07] AIR SOURCE VALVE ON (7bar)
"A0LAV101"	Q 42.0	BOOL	// ZONE1 [A0Q10] A0 LOCATOR LH X INDEX ADVANCE
"A0RAV105"	Q 42.1	BOOL	// ZONE1 [A0Q20] A0 LOCATOR RH Y INDEX ADVANCE
"A0LAV105"	Q 42.2	BOOL	// ZONE1 [A0Q10] A0 LOCATOR LH Y INDEX ADVANCE
"A0RAV109"	Q 42.3	BOOL	// ZONE1 [A0Q21] A0 LOCATOR RH Z INDEX ADVANCE
"A0LAV109"	Q 42.4	BOOL	// ZONE1 [A0Q11] A0 LOCATOR LH Z INDEX ADVANCE
"A0RAV101"	Q 42.6	BOOL	// ZONE1 [A0Q20] A0 LOCATOR RH X INDEX ADVANCE
"VATA1"	Q 43.0	BOOL	// A0SB[M06] STAGE INDICATOR AUTHORIZATION A1
"VITA1"	Q 43.1	BOOL	// A0SB[M06] STAGE INDICATOR PROHIBITION A1
"VDFA1"	Q 43.2	BOOL	// A0SB[M06] STAGE INDICATOR DEFAULT A1
"VATA2"	Q 43.5	BOOL	// A0SB[M06] STAGE INDICATOR AUTHORIZATION A2
"VITA2"	Q 43.6	BOOL	// A0SB[M06] STAGE INDICATOR PROHIBITION A2
"VDFA2"	Q 43.7	BOOL	// A0SB[M06] STAGE INDICATOR DEFAULT A2
"A0SOP"	Q 62.0	BOOL	// A0SB[M11] SAFETY LEVEL OUTPUT SOP
"A0_RFRO2"	Q 62.1	BOOL	// A0SB[M11] SAFETY LEVEL OUTPUT SOPTR
"EV7B_A0"	Q 62.3	BOOL	// EV de aire - A0
"VATB1"	Q 73.0	BOOL	// B0SB[M06] STAGE INDICATOR AUTHORIZATION B1
"VITB1"	Q 73.1	BOOL	// B0SB[M06] STAGE INDICATOR PROHIBITION B1
"VDFB1"	Q 73.2	BOOL	// B0SB[M06] STAGE INDICATOR DEFAULT B1
"VATB2"	Q 73.5	BOOL	// B0SB[M06] STAGE INDICATOR AUTHORIZATION B2
"VITB2"	Q 73.6	BOOL	// B0SB[M06] STAGE INDICATOR PROHIBITION B2
"VDFB2"	Q 73.7	BOOL	// B0SB[M06] STAGE INDICATOR DEFAULT B2
"B0SOP"	Q 92.0	BOOL	// B0SB[M11] SAFETY LEVEL OUTPUT SOP
"B0_RFRO2"	Q 92.1	BOOL	// B0SB[M11] SAFETY LEVEL OUTPUT SOPTR
"EV7B_B0"	Q 92.3	BOOL	// EV de aire - B0
"A0LAV103"	Q 107.1	BOOL	// ZONE1 [A0Q10] A0 LOCATOR LH X SLIDE ADVANCE
"A0LAV107"	Q 107.3	BOOL	// ZONE1 [A0Q10] A0 LOCATOR LH Y SLIDE ADVANCE
"A0LAV102"	Q 107.4	BOOL	// ZONE1 [A0Q10] A0 LOCATOR LH X INDEX RETURN
"A0LAV104"	Q 107.5	BOOL	// ZONE1 [A0Q10] A0 LOCATOR LH X SLIDE RETURN
"A0LAV106"	Q 107.6	BOOL	// ZONE1 [A0Q10] A0 LOCATOR LH Y INDEX RETURN
"A0LAV108"	Q 107.7	BOOL	// ZONE1 [A0Q10] A0 LOCATOR LH Y SLIDE RETURN
"A0LAV111"	Q 108.1	BOOL	// ZONE1 [A0Q11] A0 LOCATOR LH Z SLIDE ADVANCE
"A0LAV110"	Q 108.4	BOOL	// ZONE1 [A0Q11] A0 LOCATOR LH Z INDEX RETURN
"A0LAV112"	Q 108.5	BOOL	// ZONE1 [A0Q11] A0 LOCATOR LH Z SLIDE RETURN
"A0AV001"	Q 109.0	BOOL	// ZONE1 [A0Q12] A0 CLAMP ADVANCE
"A0AV003"	Q 109.1	BOOL	// ZONE1 [A0Q12] A0 L38 GAUGE SWING ADVANCE
"A0AV005"	Q 109.2	BOOL	// ZONE1 [A0Q12] A0 EJECTOR ADVANCE
"A0AV002"	Q 109.4	BOOL	// ZONE1 [A0Q12] A0 CLAMP RETURN
"A0AV004"	Q 109.5	BOOL	// ZONE1 [A0Q12] A0 L38 GAUGE SWING RETURN
"A0AV006"	Q 109.6	BOOL	// ZONE1 [A0Q12] A0 EJECTOR RETURN
"A0AV007"	Q 110.0	BOOL	// ZONE1 [A0Q13] A0 GRIPPER SHIFT 1 ADVANCE
"A0AV009"	Q 110.1	BOOL	// ZONE1 [A0Q13] A0 GRIPPER SHIFT 1 BRAKE
"A0AV011"	Q 110.2	BOOL	// ZONE1 [A0Q13] A0 GRIPPER SHIFT 2 ADVANCE
"A0AV013"	Q 110.3	BOOL	// ZONE1 [A0Q13] A0 GRIPPER LOCK 1 ADVANCE
"A0AV008"	Q 110.4	BOOL	// ZONE1 [A0Q13] A0 GRIPPER SHIFT 1 RETURN
"A0AV012"	Q 110.6	BOOL	// ZONE1 [A0Q13] A0 GRIPPER SHIFT 2 RETURN
"A0AV014"	Q 110.7	BOOL	// ZONE1 [A0Q13] A0 GRIPPER LOCK 1 RETURN
"A0RAV103"	Q 157.1	BOOL	// ZONE1 [A0Q20] A0 LOCATOR RH X SLIDE ADVANCE
"A0RAV107"	Q 157.3	BOOL	// ZONE1 [A0Q20] A0 LOCATOR RH Y SLIDE ADVANCE
"A0RAV102"	Q 157.4	BOOL	// ZONE1 [A0Q20] A0 LOCATOR RH X INDEX RETURN
"A0RAV104"	Q 157.5	BOOL	// ZONE1 [A0Q20] A0 LOCATOR RH X SLIDE RETURN
"A0RAV106"	Q 157.6	BOOL	// ZONE1 [A0Q20] A0 LOCATOR RH Y INDEX RETURN
"A0RAV108"	Q 157.7	BOOL	// ZONE1 [A0Q20] A0 LOCATOR RH Y SLIDE RETURN
"A0RAV111"	Q 158.1	BOOL	// ZONE1 [A0Q21] A0 LOCATOR RH Z SLIDE ADVANCE
"A0RAV110"	Q 158.4	BOOL	// ZONE1 [A0Q21] A0 LOCATOR RH Z INDEX RETURN
"A0RAV112"	Q 158.5	BOOL	// ZONE1 [A0Q21] A0 LOCATOR RH Z SLIDE RETURN
"A0AV015"	Q 159.0	BOOL	// ZONE1 [A0Q22] A0 GRIPPER LOCK 2 ADVANCE
"A0AV017"	Q 159.1	BOOL	// ZONE1 [A0Q22] A0 MODEL CHANGE 1 ADVANCE
"A0AV019"	Q 159.2	BOOL	// ZONE1 [A0Q22] A0 MODEL CHANGE 2 ADVANCE
"A0AV016"	Q 159.4	BOOL	// ZONE1 [A0Q22] A0 GRIPPER LOCK 2 RETURN
"A0AV018"	Q 159.5	BOOL	// ZONE1 [A0Q22] A0 MODEL CHANGE 1 RETURN
"A0AV020"	Q 159.6	BOOL	// ZONE1 [A0Q22] A0 MODEL CHANGE 2 RETURN
"B0LAV101"	Q 207.0	BOOL	// ZONE1 [B0Q10] B0 LOCATOR LH X INDEX ADVANCE
"B0LAV103"	Q 207.1	BOOL	// ZONE1 [B0Q10] B0 LOCATOR LH X SLIDE ADVANCE
"B0LAV105"	Q 207.2	BOOL	// ZONE1 [B0Q10] B0 LOCATOR LH Y INDEX ADVANCE
"B0LAV107"	Q 207.3	BOOL	// ZONE1 [B0Q10] B0 LOCATOR LH Y SLIDE ADVANCE
"B0LAV102"	Q 207.4	BOOL	// ZONE1 [B0Q10] B0 LOCATOR LH X INDEX RETURN
"B0LAV104"	Q 207.5	BOOL	// ZONE1 [B0Q10] B0 LOCATOR LH X SLIDE RETURN
"B0LAV106"	Q 207.6	BOOL	// ZONE1 [B0Q10] B0 LOCATOR LH Y INDEX RETURN
"B0LAV108"	Q 207.7	BOOL	// ZONE1 [B0Q10] B0 LOCATOR LH Y SLIDE RETURN
"B0LAV109"	Q 208.0	BOOL	// ZONE1 [B0Q11] B0 LOCATOR LH Z INDEX ADVANCE
"B0LAV111"	Q 208.1	BOOL	// ZONE1 [B0Q11] B0 LOCATOR LH Z SLIDE ADVANCE
"B0LAV110"	Q 208.4	BOOL	// ZONE1 [B0Q11] B0 LOCATOR LH Z INDEX RETURN
"B0LAV112"	Q 208.5	BOOL	// ZONE1 [B0Q11] B0 LOCATOR LH Z SLIDE RETURN
"B0AV001"	Q 209.0	BOOL	// ZONE1 [B0Q12] B0 CLAMP ADVANCE
"B0AV003"	Q 209.1	BOOL	// ZONE1 [B0Q12] B0 L38 GAUGE SWING ADVANCE
"B0AV005"	Q 209.2	BOOL	// ZONE1 [B0Q12] B0 EJECTOR ADVANCE
"B0AV007"	Q 209.3	BOOL	// ZONE1 [B0Q12] B0 OG SHIFT ADVANCE
"B0AV002"	Q 209.4	BOOL	// ZONE1 [B0Q12] B0 CLAMP RETURN
"B0AV004"	Q 209.5	BOOL	// ZONE1 [B0Q12] B0 L38 GAUGE SWING RETURN
"B0AV006"	Q 209.6	BOOL	// ZONE1 [B0Q12] B0 EJECTOR RETURN
"B0AV008"	Q 209.7	BOOL	// ZONE1 [B0Q12] B0 OG SHIFT RETURN
"B0AV009"	Q 210.0	BOOL	// ZONE1 [B0Q13] B0 OG LOCK ADVANCE
"B0AV011"	Q 210.1	BOOL	// ZONE1 [B0Q13] B0 GRIPPER LOCK ADVANCE
"B0AV013"	Q 210.2	BOOL	// ZONE1 [B0Q13] B0 MODEL CHANGE 1 ADVANCE
"B0AV010"	Q 210.4	BOOL	// ZONE1 [B0Q13] B0 OG LOCK RETURN
"B0AV012"	Q 210.5	BOOL	// ZONE1 [B0Q13] B0 GRIPPER LOCK RETURN
"B0AV014"	Q 210.6	BOOL	// ZONE1 [B0Q13] B0 MODEL CHANGE 1 RETURN
"B0RAV101"	Q 257.0	BOOL	// ZONE1 [B0Q20] B0 LOCATOR RH X INDEX ADVANCE
"B0RAV103"	Q 257.1	BOOL	// ZONE1 [B0Q20] B0 LOCATOR RH X SLIDE ADVANCE
"B0RAV105"	Q 257.2	BOOL	// ZONE1 [B0Q20] B0 LOCATOR RH Y INDEX ADVANCE
"B0RAV107"	Q 257.3	BOOL	// ZONE1 [B0Q20] B0 LOCATOR RH Y SLIDE ADVANCE
"B0RAV102"	Q 257.4	BOOL	// ZONE1 [B0Q20] B0 LOCATOR RH X INDEX RETURN
"B0RAV104"	Q 257.5	BOOL	// ZONE1 [B0Q20] B0 LOCATOR RH X SLIDE RETURN
"B0RAV106"	Q 257.6	BOOL	// ZONE1 [B0Q20] B0 LOCATOR RH Y INDEX RETURN
"B0RAV108"	Q 257.7	BOOL	// ZONE1 [B0Q20] B0 LOCATOR RH Y SLIDE RETURN
"B0RAV109"	Q 258.0	BOOL	// ZONE1 [B0Q21] B0 LOCATOR RH Z INDEX ADVANCE
"B0RAV111"	Q 258.1	BOOL	// ZONE1 [B0Q21] B0 LOCATOR RH Z SLIDE ADVANCE
"B0RAV110"	Q 258.4	BOOL	// ZONE1 [B0Q21] B0 LOCATOR RH Z INDEX RETURN
"B0RAV112"	Q 258.5	BOOL	// ZONE1 [B0Q21] B0 LOCATOR RH Z SLIDE RETURN
"B0AV015"	Q 259.0	BOOL	// ZONE1 [B0Q22] B0 MODEL CHANGE 2 ADVANCE
"B0AV017"	Q 259.1	BOOL	// ZONE1 [B0Q22] B0 MODEL CHANGE 3 ADVANCE
"B0AV016"	Q 259.4	BOOL	// ZONE1 [B0Q22] B0 MODEL CHANGE 2 RETURN
"B0AV018"	Q 259.5	BOOL	// ZONE1 [B0Q22] B0 MODEL CHANGE 3 RETURN
"D0_OP1VAT"	Q 271.0	BOOL	// D0SB[M06] WORK AUTORISATION LAMP 1(GREEN)
"D0_OP1VIT"	Q 271.1	BOOL	// D0SB[M06] WORK PROHIBITION LAMP 1 (RED)
"D0_OP1VDF"	Q 271.2	BOOL	// D0SB[M06] DEFAULT LAMP 1 (ORANGE)
"C0_OP1VDF"	Q 271.5	BOOL	// D0SB[M06] C0 DEFAULT LAMP 1 (VERDE)
"C0_OP1BZZ"	Q 271.6	BOOL	// D0SB[M06] C0 DEFAULT BUZZER
"D0_RFRO1"	Q 290.0	BOOL	// D0SB[M11] SAFETY COMMON 3
"D0_RFRO2"	Q 290.1	BOOL	// D0SB[M11] SAFETY COMMON 4
"D0_RFRO3"	Q 290.2	BOOL	// D0SB[M11] SAFETY COMMON 5
"EV7B_D0"	Q 290.3	BOOL	// EV de aire - D0
"D01EAPL1"	Q 300.0	BOOL	// ZONE1 [D0A1] PIN CLAMP 1 ADVANCE
"D01ERPL1"	Q 300.1	BOOL	// ZONE1 [D0A1] PIN CLAMP 1 RETURN
"D01EASR2"	Q 300.2	BOOL	// ZONE1 [D0A1] CLAMP 2 ADVANCE
"D01ERSR2"	Q 300.3	BOOL	// ZONE1 [D0A1] CLAMP 2 RETURN
"D0_VVAL"	Q 304.0	BOOL	// Habilitacion de 24V Valvulas CPX D0DTS1
"D0EVCPX"	Q 304.1	BOOL	// Electrovalvula CPX D0DTS1
"A01EASR1"	Q 400.0	BOOL	// ZONE1 [A0A1] CLAMP 1 ADVANCE
"A01ERSR1"	Q 400.1	BOOL	// ZONE1 [A0A1] CLAMP 1 RETURN
"A0_VVAL"	Q 404.0	BOOL	// Habilitacion de 24V Valvulas CPX A0DTS1
"A0EVCPX"	Q 404.1	BOOL	// electrovalvula CPX A0DTS1
"B01EASR1"	Q 450.0	BOOL	// ZONE1 [B0A1] CLAMP 1 AVANCE
"B01ERSR1"	Q 450.1	BOOL	// ZONE1 [B0A1] CLAMP 1 RETROCESO
"B01EASR2"	Q 450.2	BOOL	// ZONE1 [B0A1] CLAMP 2 AVANCE
"B01ERSR2"	Q 450.3	BOOL	// ZONE1 [B0A1] CLAMP 2 RETROCESO
"B01EAPL3"	Q 450.4	BOOL	// ZONE1 [B0A1] PILOTO 3 AVANCE
"B01ERPL3"	Q 450.5	BOOL	// ZONE1 [B0A1] PILOTO 3 RETROCESO
"B01EAPL4"	Q 450.6	BOOL	// ZONE1 [B0A1] PILOTO 4 AVANCE
"B01ERPL4"	Q 450.7	BOOL	// ZONE1 [B0A1] PILOTO 4 RETROCESO
"B01EFRPL31"	Q 451.0	BOOL	// ZONE1 [B0A1] TRABA DE VASTAGO PL31
"B01EFRPL32"	Q 451.1	BOOL	// ZONE1 [B0A1] TRABA DE VASTAGO PL32
"B01EFRPL41"	Q 451.2	BOOL	// ZONE1 [B0A1] TRABA DE VASTAGO PL41
"B01EFRPL42"	Q 451.3	BOOL	// ZONE1 [B0A1] TRABA DE VASTAGO PL42
"B01EASR6"	Q 451.4	BOOL	// ZONE1 [B0A1] CLAMP 5 AVANCE
"B01ERSR6"	Q 451.5	BOOL	// ZONE1 [B0A1] CLAMP 5 RETROCESO
"B01_VVAL"	Q 454.0	BOOL	// Habilitacion de 24V Valvulas CPX B0DTS1
"B01EVCPX"	Q 454.1	BOOL	// Electrovalvula CPX B0DTS1
"B02EAPL1"	Q 500.0	BOOL	// ZONE1 [B0A1] GRIPPER SLIDE 1 ADVANCE
"B02ERPL1"	Q 500.1	BOOL	// ZONE1 [B0A1] GRIPPER SLIDE 1 RETURN
"B02EAPL2"	Q 500.2	BOOL	// ZONE1 [B0A1] GRIPPER SLIDE 2 ADVANCE
"B02ERPL2"	Q 500.3	BOOL	// ZONE1 [B0A1] GRIPPER SLIDE 2 RETURN
"B02EAPL3"	Q 500.4	BOOL	// ZONE1 [B0A1] GRIPPER PIN CLAMP 1 ADVANCE
"B02ERPL3"	Q 500.5	BOOL	// ZONE1 [B0A1] GRIPPER PIN CLAMP 1 RETURN
"B02EAPL4"	Q 500.6	BOOL	// ZONE1 [B0A1] GRIPPER PIN CLAMP 1 ADVANCE
"B02ERPL4"	Q 500.7	BOOL	// ZONE1 [B0A1] GRIPPER PIN CLAMP 1 RETURN
"B02EASR5"	Q 501.0	BOOL	// ZONE1 [B0A1] GRIPPER CLAMP 5 ADVANCE
"B02ERSR5"	Q 501.1	BOOL	// ZONE1 [B0A1] GRIPPER CLAMP 5 RETURN
"B02EASR6"	Q 501.2	BOOL	// ZONE1 [B0A1] GRIPPER CLAMP 6 ADVANCE
"B02ERSR6"	Q 501.3	BOOL	// ZONE1 [B0A1] GRIPPER CLAMP 6 RETURN
"B02EAPL7"	Q 501.4	BOOL	// ZONE1 [B0A1] GRIPPER PIN CLAMP 7 ADVANCE
"B02ERPL7"	Q 501.5	BOOL	// ZONE1 [B0A1] GRIPPER PIN CLAMP 7 RETURN
"B02EASR8"	Q 501.6	BOOL	// ZONE1 [B0A1] GRIPPER CLAMP 8 ADVANCE
"B02ERSR8"	Q 501.7	BOOL	// ZONE1 [B0A1] GRIPPER CLAMP 8 RETURN
"B02_VVAL"	Q 506.0	BOOL	// Habilitacion de 24V Valvulas CPX B0DTS2
"B02EVCPX"	Q 506.1	BOOL	// Electrovalvula CPX B0DTS2
"LGSB_M4_R1"	Q 550.0	BOOL	// [LGSB.M04]: RESERVA
"LGSB_M4_R2"	Q 550.1	BOOL	// [LGSB.M04]: RESERVA
"LGSB_M4_R3"	Q 550.2	BOOL	// [LGSB.M04]: RESERVA
"LGSB_M4_R4"	Q 550.3	BOOL	// [LGSB.M04]: RESERVA
"LGSB_M4_R5"	Q 550.4	BOOL	// [LGSB.M04]: RESERVA
"LGSB_M4_R6"	Q 550.5	BOOL	// [LGSB.M04]: RESERVA
"LGSB_M4_R7"	Q 550.6	BOOL	// [LGSB.M04]: RESERVA
"LGSB_M4_R8"	Q 550.7	BOOL	// [LGSB.M04]: RESERVA
"LG1VAT"	Q 551.0	BOOL	// [LGSB.M06]: LG1 WORK AUTORISATION LAMP 1 (GREEN)
"LG1VIT"	Q 551.1	BOOL	// [LGSB.M06]: LG1 WORK PROHIBITION LAMP 1 (RED)
"LG1VDF"	Q 551.2	BOOL	// [LGSB.M06]: LG1 DEFAULT LAMP 1 (ORANGE)
"LGSB_M6_R1"	Q 551.3	BOOL	// [LGSB.M06]: RESERVA
"LGSB_M6_R2"	Q 551.4	BOOL	// [LGSB.M06]: RESERVA
"LGSB_M6_R3"	Q 551.5	BOOL	// [LGSB.M06]: RESERVA
"LGSB_M6_R4"	Q 551.6	BOOL	// [LGSB.M06]: RESERVA
"LGSB_M6_R5"	Q 551.7	BOOL	// [LGSB.M06]: RESERVA
"LGRFRO1"	Q 572.0	BOOL	// [LGSB.M11]: LG SAFETY COMMON 3 (F0SOP)
"LGRFRO2"	Q 572.1	BOOL	// [LGSB.M11]: LG SAFETY COMMON 4 (Z2ES)
"LGRFRO3"	Q 572.2	BOOL	// [LGSB.M11]: LG SAFETY COMMON 5 (F0)
"LGSB_M11_R1"	Q 572.3	BOOL	// [LGSB.M11]: RESERVA
"LGEASR1"	Q 600.0	BOOL	// [LGIM1.LGS11]: LG: EV AVANCE SR1
"LGERSR1"	Q 600.1	BOOL	// [LGIM1.LGS11]: LG: EV RETROCESO SR1
"LGEAPLB"	Q 600.2	BOOL	// [LGIM1.LGS11]: LG: EV AVANCE CILINDRO CAMBIO DE MASA
"LGERPLB"	Q 600.3	BOOL	// [LGIM1.LGS11]: LG: EV RETROCESO CILINDRO CAMBIO DE MASA
"LGEASR2"	Q 600.4	BOOL	// [LGIM1.LGS11]: LG: EV AVANCE SR2
"LGERSR2"	Q 600.5	BOOL	// [LGIM1.LGS11]: LG: EV RETROCESO SR2
"LGEASR3"	Q 600.6	BOOL	// [LGIM1.LGS11]: LG: EV AVANCE SR3
"LGERSR3"	Q 600.7	BOOL	// [LGIM1.LGS11]: LG: EV RETROCESO SR3
"LGEASR4"	Q 601.0	BOOL	// [LGIM1.LGS11]: LG: EV AVANCE SR4
"LGERSR4"	Q 601.1	BOOL	// [LGIM1.LGS11]: LG: EV RETROCESO SR4
"LGEAVU5"	Q 601.2	BOOL	// [LGIM1.LGS11]: LG: EV AVANCE VU5
"LGERVU5"	Q 601.3	BOOL	// [LGIM1.LGS11]: LG: EV RETROCESO VU5
"LGEAVU6"	Q 601.4	BOOL	// [LGIM1.LGS11]: LG: EV AVANCE VU6
"LGERVU6"	Q 601.5	BOOL	// [LGIM1.LGS11]: LG: EV RETROCESO VU6
"LGCAM1"	Q 607.0	BOOL	// [LGIM2.LGDM21]: LG: COMANDO AVANÇO MOTOR M1
"LGCRM1"	Q 607.1	BOOL	// [LGIM2.LGDM21]: LG: COMANDO RECUO MOTOR M1
"LGMOTRAZ"	Q 607.3	BOOL	// Reset modulo motor LG
"LDEASR1"	Q 620.0	BOOL	// [LDIM1.LDS11]: LD: EV AVANCE SR1
"LDERSR1"	Q 620.1	BOOL	// [LDIM1.LDS11]: LD: EV RETROCESO SR1
"LDEASR2"	Q 620.2	BOOL	// [LDIM1.LDS11]: LD: EV AVANCE SR2
"LDERSR2"	Q 620.3	BOOL	// [LDIM1.LDS11]: LD: EV RETROCESO SR2
"LDEAVU3"	Q 620.4	BOOL	// [LDIM1.LDS11]: LD: EV AVANCE VU3
"LDERVU3"	Q 620.5	BOOL	// [LDIM1.LDS11]: LD: EV RETROCESO VU3
"LDEASR4"	Q 620.6	BOOL	// [LDIM1.LDS11]: LD: EV AVANCE SR4
"LDERSR4"	Q 620.7	BOOL	// [LDIM1.LDS11]: LD: EV RETROCESO SR4
"LDEASR5"	Q 621.0	BOOL	// [LDIM1.LDS12]: LD: EV AVANCE SR5
"LDERSR5"	Q 621.1	BOOL	// [LDIM1.LDS12]: LD: EV RETROCESO SR5
"LDEAVU6"	Q 621.2	BOOL	// [LDIM1.LDS12]: LD: EV AVANCE VU6
"LDERVU6"	Q 621.3	BOOL	// [LDIM1.LDS12]: LD: EV RETROCESO VU6
"LDEAVU7"	Q 621.4	BOOL	// [LDIM1.LDS12]: LD: EV AVANCE VU7
"LDERVU7"	Q 621.5	BOOL	// [LDIM1.LDS12]: LD: EV RETROCESO VU7
"LDCAM1"	Q 627.0	BOOL	// [LDIM2.LDDM21]: LD: COMANDO AVANÇO MOTOR M1
"LDCRM1"	Q 627.1	BOOL	// [LDIM2.LDDM21]: LD: COMANDO RECUO MOTOR M1
"LDMOTRAZ"	Q 627.3	BOOL	// Reset modulo motor LD
"LDSB_M3_R5SB_M4_R1"	Q 630.0	BOOL	// [LDSB.M04]: RESERVA
"LDSB_M3_R5SB_M4_R2"	Q 630.1	BOOL	// [LDSB.M04]: RESERVA
"LDSB_M3_R5SB_M4_R3"	Q 630.2	BOOL	// [LDSB.M04]: RESERVA
"LDSB_M3_R5SB_M4_R4"	Q 630.3	BOOL	// [LDSB.M04]: RESERVA
"LDSB_M3_R5SB_M4_R5"	Q 630.4	BOOL	// [LDSB.M04]: RESERVA
"LDSB_M3_R5SB_M4_R6"	Q 630.5	BOOL	// [LDSB.M04]: RESERVA
"LDSB_M3_R5SB_M4_R7"	Q 630.6	BOOL	// [LDSB.M04]: RESERVA
"LDSB_M3_R5SB_M4_R8"	Q 630.7	BOOL	// [LDSB.M04]: RESERVA
"LD1VAT"	Q 631.0	BOOL	// [LDSB.M06]: LD1 WORK AUTORISATION LAMP 1 (GREEN)
"LD1VIT"	Q 631.1	BOOL	// [LDSB.M06]: LD1 WORK PROHIBITION LAMP 1 (RED)
"LD1VDF"	Q 631.2	BOOL	// [LDSB.M06]: LD1 DEFAULT LAMP 1 (ORANGE)
"LDSB_M3_R5SB_M6_R1"	Q 631.3	BOOL	// [LDSB.M06]: RESERVA
"LDSB_M3_R5SB_M6_R2"	Q 631.4	BOOL	// [LDSB.M06]: RESERVA
"LDSB_M3_R5SB_M6_R3"	Q 631.5	BOOL	// [LDSB.M06]: RESERVA
"LDSB_M3_R5SB_M6_R4"	Q 631.6	BOOL	// [LDSB.M06]: RESERVA
"LDSB_M3_R5SB_M6_R5"	Q 631.7	BOOL	// [LDSB.M06]: RESERVA
"LDRFRO1"	Q 660.0	BOOL	// [LDSB.M11]: LDSAFETY COMMON 3 (G0SOP)
"LDRFRO2"	Q 660.1	BOOL	// [LDSB.M11]: LD SAFETY COMMON 4 (Z2ES)
"LDRFRO3"	Q 660.2	BOOL	// [LDSB.M11]: LD SAFETY COMMON 5 (G0)
"LDSB_M11_R1"	Q 660.3	BOOL	// [LDSB.M11]: RESERVA
"TP"	SFB 3	SFB 3	// Generate a Pulse
"TON"	SFB 4	SFB 4	// Generate an On Delay
"TOF"	SFB 5	SFB 5	// Generate an Off Delay
"RDREC"	SFB 52	SFB 52	// Read a Process Data Record
"WRREC"	SFB 53	SFB 53	// Write a Process Data Record
"RALRM"	SFB 54	SFB 54	// Receive Alarm Data
"SET_CLK"	SFC 0	SFC 0	// Set System Clock
"READ_CLK"	SFC 1	SFC 1	// Read System Clock
"RD_SINFO"	SFC 6	SFC 6	// Read OB Start Information
"DPRD_DAT"	SFC 14	SFC 14	// Read Consistent Data of a Standard DP Slave
"DPWR_DAT"	SFC 15	SFC 15	// Write Consistent Data to a Standard DP Slave
"BLKMOV"	SFC 20	SFC 20	// Copy Variables
"FILL"	SFC 21	SFC 21	// Initialize a Memory Area
"TEST_DB"	SFC 24	SFC 24	// Test Data Block
"DIS_AIRT"	SFC 41	SFC 41	// Delay the Higher Priority Interrupts and Asynchronous Errors
"EN_AIRT"	SFC 42	SFC 42	// Enable Higher Priority Interrupts and Asynchronous Errors
"STP"	SFC 46	SFC 46	// Change the CPU to STOP
"RDSYSST"	SFC 51	SFC 51	// Read a System Status List or Partial List
"WR_REC"	SFC 58	SFC 58	// Write Data Record
"RD_REC"	SFC 59	SFC 59	// Read a Data Record
"TIME_TCK"	SFC 64	SFC 64	// Read the System Time
"GEO_LOG"	SFC 70	SFC 70	// Determine Logical Address
"READ_DBL"	SFC 83	SFC 83	// Read Data Block out of Load Memory
"WRIT_DBL"	SFC 84	SFC 84	// Write Data Block in Load Memory
"DEL_SI"	SFC 106	SFC 106	// Deleting Dynamically Assigned System Instances
"ALARM_DQ"	SFC 107	SFC 107	// Creating Acknowledgeable Block-related Message
"ALARM_D"	SFC 108	SFC 108	// Creating Acknowledged Block-related Message
"lien_Sec"	UDT 1507	UDT 1507	// Table de 6 mots commun aux FB ZONE_PORTE, ZONE_RSEC, ZONE_MODES
"IN_FONC"	UDT 1520	UDT 1520	// Gestion de la Fonction In du variateur de Manutention Standard (BF_FONC_VAR2)
"PILOTAGE"	UDT 1521	UDT 1521	// Gestion de la Fonction Pilotage du variateur de Manutention Standard (FONC_VAR2)
"OUT_FONC"	UDT 1522	UDT 1522	// Gestion de la Fonction Out du variateur de Manutention Standard (BF_FONC_VAR2)
"Lien_Pup"	UDT 1988	UDT 1988	// ZONE : Traitement des Modes pupitre cde manuelle
"SL_IHM"	UDT 1999	UDT 1999
"Lien_Ilot"	UDT 2004	UDT 2004	// ILOT : Gestion info lié à l'installation (ILOT)
"MOT_FONC_MP"	UDT 2041	UDT 2041	// INFO CONTROL OF A MOVEMENT (BF_MOUVMP1)
"MOT_FONC"	UDT 2042	UDT 2042	// Gestion info d'un mouvement (BF_MOUV2P1,BF_MVSE2P1, BF_RB_COD_PREH_API)
"FONC"	UDT 2047	UDT 2047	// Gestion info d'un relais en double canal (BF_FILERIE1, BF_SEC_COM)
"CDIV_AOL"	VAT 1	
"IIT_"	VAT 2	
"RFID"	VAT 3	
"VAT_4"	VAT 4	
"SIPTOL_A0L"	VAT 5	
"SIPTOL_D0R"	VAT 6	
"SIPTOL_ACQ_A0L"	VAT 7	
"SIPTOL"	VAT 8	
"SIPTOL_D0R_simple"	VAT 9	
"IIT_1"	VAT 10	
"VAT_11"	VAT 11	
"SIPTOL_D0R_LEO"	VAT 12	
"B0_LCB"	VAT 13	
END_SYMBOL_TABLE
